REGION Network 4: Block description — Section 3.6 to 4
   // ▂▂▂▂▂▂▂▂▂▂▂▂▂▂▂▂▂▂▂▂▂▂▂▂▂▂▂▂▂▂▂▂▂▂▂▂▂▂▂▂▂▂▂▂
   // 3.6     Operating modes
   // 
   // 
   // This module FC11001_StdDevValveIsol supports various operating modes:
   // 
   //    •   Automatic/manual mode
   // 
   //    •   Interlock bypass mode
   // 
   //    •   Simulation mode
   // 
   //    •   Remote/local mode
   // 
   //    •   Faceplate disabled mode
   // 
   // Examining these in turn:   
   // 
   // 
   // 
   // ▁▁▁▁▁▁▁▁▁▁▁▁▁▁▁▁▁▁▁▁▁▁▁▁▁▁▁▁▁▁▁▁▁▁▁▁▁▁▁▁▁▁▁▁
   // 3.6.1    Automatic and manual modes
   // 
   // 
   // Under normal operation, the valve is in automatic mode and is controlled directly by the 
   // Controller software (usually, sequential or continuous logic); however, it is possible for the 
   // operator to take direct control of the valve by switching it to manual mode.
   // 
   // If manual mode is active, the valve will open and close directly at the command of the operator 
   // and will ignore any automatic mode open and close requests.
   // 
   // If the valve is operating under automatic mode, the manual open/close request follows that of 
   // the automatic mode; this ensures that the valve remains in the same state when initially 
   // switched from automatic mode to manual mode, referred to as bumpless transfer. This approach 
   // minimises any disturbance to the process should the valve be inadvertently switched to manual 
   // mode.
   // 
   // The following data points are associated with automatic/manual mode:
   // 
   //  DATA STRUCTURE    UT11001_St_DevValveIsol
   //  ――――――――――――――――――――――――――――――――――――――――――
   //  SIGNAL         FUNCTION               TYPE     DETAILS
   //  ――――――――――――――――――――――――――――――――――――――――――
   //  CONFIG_MAN_DIS     Prevents manual mode being       Bool  1 = no manual mode
   //            activated under all circumstances            0 = manual permitted
   //  ――――――――――――――――――――――――――――――――――――――――――
   // 
   //  DATA STRUCTURE    UT31001_Dy_DevValveIsol
   //  ――――――――――――――――――――――――――――――――――――――――――
   //  SIGNAL         FUNCTION               TYPE     DETAILS
   //  ――――――――――――――――――――――――――――――――――――――――――
   //  Mode_AutMan     Identifies the operating mode of     Bool  1 = automatic mode
   //            the valve.                   0 = manual mode
   // 
   //  ctrl_Aut_OpenClose Causes the valve to open and close     Bool  1 = open the valve
   //            if automatic mode is active            0 = close the valve
   // 
   //  ctrl_Man_OpenClose  Causes the valve to open and close     Bool  1 = open the valve
   //            if manual mode is active             0 = close the valve
   // 
   //  status_Aut      The valve is in automatic mode      Bool  1 = auto mode
   //                                  0 = no in auto
   // 
   //  status_Man       The valve is in manual mode     Bool  1 = manual mode
   //                                  0 = no in manual
   //  ――――――――――――――――――――――――――――――――――――――――――
   // 
   // Manual mode can only be activated by the operator via a faceplate available at the supervisory 
   // system (SCADA/HMI). 
   // 
   // 
   // 
   // ▁▁▁▁▁▁▁▁▁▁▁▁▁▁▁▁▁▁▁▁▁▁▁▁▁▁▁▁▁▁▁▁▁▁▁▁▁▁▁▁▁▁▁▁
   // 3.6.2    Interlock bypass mode
   // 
   // 
   // All interlock signals (TRIP, INTERLOCK or PERMISSIVE) can be overridden (bypassed). The bypass 
   // signal is a single signal that, if active, overrides and deactivates any TRIP, INTERLOCK or 
   // PERMISSIVE signal that may have been activated.
   // 
   // It is possible to permanently disable the bypass mode for any given valve (preventing the 
   // operator from activating it).
   // 
   // The following data points are associated with the bypass mode:
   // 
   //  DATA STRUCTURE    UT11001_St_DevValveIsol
   //  ――――――――――――――――――――――――――――――――――――――――――
   //  SIGNAL       FUNCTION                TYPE     DETAILS
   //  ――――――――――――――――――――――――――――――――――――――――――
   //  CONFIG_BYPASS_DIS    Prevents bypass mode being      Bool     1 = no bypass mode
   //             activated under all circumstances         0 = bypass permitted
   //  ――――――――――――――――――――――――――――――――――――――――――
   // 
   //  DATA STRUCTURE    UT31001_Dy_DevValveIsol
   //  ――――――――――――――――――――――――――――――――――――――――――
   //  SIGNAL         FUNCTION                TYPE     DETAILS
   //  ――――――――――――――――――――――――――――――――――――――――――
   //  mode_BypassOn   Activates bypass mode, if active, any    Bool     1 = bypass mode on
   //            TRIP, INTERLOCK or PERMISSIVE signal          0 = bypass mode off
   //            will be ignored
   // 
   //  status_BypassOn   Status indication, shows if bypass      Bool     1 = bypass active
   //            mode is active                 0 = bypass inactive
   //  ――――――――――――――――――――――――――――――――――――――――――
   // 
   // Bypass mode can only be activated by the operator usually via a faceplate available at the 
   // supervisory system (SCADA/HMI), alternatively it may be via some form of hardwired signal such 
   // as a key-switch &c. 
   // 
   // If bypass mode is disabled (configuration signal CONFIG_BYPASS_DIS is set to 1), then the bypass 
   // mode cannot be turned on under any circumstances, the option will be greyed out on the 
   // supervisory system faceplate and the module will constantly reset the mode_BypassOn signal.  
   // 
   // 
   // 
   // ▁▁▁▁▁▁▁▁▁▁▁▁▁▁▁▁▁▁▁▁▁▁▁▁▁▁▁▁▁▁▁▁▁▁▁▁▁▁▁▁▁▁▁▁
   // 3.6.3    Simulation mode
   // 
   // 
   // The module can be switched to a simulation mode, in which the position feedback for the valve 
   // is replaced by simulated signals specified by the operator. 
   // 
   // Simulation mode is generally used during testing, but can also be applied in a process 
   // environment if a fault condition is detected; this scenario allows the plant to continue operating 
   // (albeit under some degree of manual control) until the valve is repaired or replaced.
   // 
   // The following data points are associated with the simulation mode:
   // 
   //  DATA STRUCTURE    UT11001_St_DevValveIsol
   //  ――――――――――――――――――――――――――――――――――――――――――
   //  SIGNAL       FUNCTION                TYPE     DETAILS
   //  ――――――――――――――――――――――――――――――――――――――――――
   //  CONFIG_SIM_DIS     Prevents simulation mode being     Bool     1 = no sim mode
   //             activated under all circumstances         0 = sim permitted
   //  ――――――――――――――――――――――――――――――――――――――――――
   // 
   //  DATA STRUCTURE    UT31001_Dy_DevValveIsol
   //  ――――――――――――――――――――――――――――――――――――――――――
   //  SIGNAL         FUNCTION                TYPE     DETAILS
   //  ――――――――――――――――――――――――――――――――――――――――――
   //  mode_SimOn      Activates simulation mode, if active, the   Bool     1 = sim mode on
   //            position feedback will be specified by         0 = sim mode off
   //            mode_SimValue      
   //  mode_SimValue    Specifies the type of simulated position     Int     0 = no feedback
   //            feedback in use                  1 = permanently open
   //                                      2 = permanently closed
   //                                      3 = follow demand
   // 
   //  status_SimOn     Status indication, shows if simulation     Bool     1 = sim active
   //            mode is active                 0 = sim inactive
   //  ――――――――――――――――――――――――――――――――――――――――――
   // 
   // Simulation mode can only be activated by the operator via a faceplate available at the 
   // supervisory system (SCADA/HMI).
   // 
   // If simulation mode is activated, the position feedback for the valve is forced to one of four 
   // states specified by the mode_SimValue variable (this is an enumerated variable):
   // 
   //  ――――――――――――――――――――――――――――――――――――――――――
   //  mode_SimValue  DESCRIPTION               FBK_OPEN FBK_CLOSED
   //  ――――――――――――――――――――――――――――――――――――――――――
   //      0        Permanently disables all position feedback    0     0
   //             (irrespective of any valve position)
   // 
   //      1        Permanently sets valve position to open         1     0
   //             (irrespective of any valve position)
   // 
   //      2        Permanently sets valve position to closed      0     1
   //             (irrespective of any valve position)
   // 
   //      3        Position feedback follows the requested        1/0    0/1
   //             state of the valve              (if valve is open/closed)
   //  ――――――――――――――――――――――――――――――――――――――――――
   // 
   // The mode_SimValue is restricted to the range 0-3.
   // 
   // If simulation mode is disabled (configuration signal CONFIG_SIM_DIS is set to 1), then the 
   // simulation mode cannot be turned on under any circumstances, the option will be greyed out on 
   // the supervisory system faceplate and the module will constantly reset the mode_SimOn signal.
   // 
   // If simulation mode is permitted (CONFIG_SIM_DIS = 0), then setting mode_SimOn to 1 will activate 
   // simulation mode and the any position feedback signals (connected to FBK_OPEN and 
   // FBK_CLOSED) will be overridden according to the value stored in mode_SimValue (see Table above).
   // 
   // The operator can set and adjust the simulation value (mode_SimValue) from the instrument 
   // faceplate on the supervisory system. The simulation value can be adjusted at any time by the 
   // operator (even if simulation mode has not been activated), but will not be applied until 
   // simulation mode is turned on (mode_SimOn = 1). 
   // 
   // If simulation mode is completely disabled (CONFIG_SIM_DIS is set to 1) then the operator will not 
   // be able to adjust the simulated value (mode_SimValue will be greyed out on the faceplate).
   // 
   // 
   // 
   // ▁▁▁▁▁▁▁▁▁▁▁▁▁▁▁▁▁▁▁▁▁▁▁▁▁▁▁▁▁▁▁▁▁▁▁▁▁▁▁▁▁▁▁▁
   // 3.6.4     Remote/local mode
   // 
   // Remote and local operating modes refer to the supervisory system that has control of the 
   // device (i.e. which system can write to the device and change the operating mode of the 
   // device). 
   // 
   // This type of mode is usual present where a plant has a remote central control location (a control 
   // room) that normally controls the device (remote control), but also has a field panel with a local 
   // HMI that an operator in the field can select to take over control of the device (local control) for 
   // maintenance purposes.
   // 
   // The modes are as follows (and are mutually exclusive, only one will be active):
   // 
   //    Remote        Only the remote system in the control room can 
   //                 control the device
   // 
   //    Local            A local system has taken control of the device and the remote 
   //                 system can no longer issue commands to it
   // 
   //    Remote/local disabled   The system does not use remote/local modes and any 
   //      (ALL mode)     supervisory system can issue commands to the device 
   //  
   // Remote/local control is generally handled by the supervisory systems themselves; however, the 
   // supervisory systems need a storage area per device to record which mode that device is in, local 
   // control is often activated by a panel key-switch, that changes the state of several devices from 
   // remote to local (usually all the devices controlled by the local panel).
   // 
   // The module simply identifies the remote/local mode from the mode signals and configuration 
   // signals provided to the module.
   // 
   // For systems that do not use remote/local modes (any supervisory system can control the device, 
   // or control is determined by operator privileges), the remote/local modes can be disabled 
   // (CONFIG_RL_EN is set to zero) and the device is effectively in ALL mode (any system can 
   // control the device).
   // 
   // If remote/local operation is in use, the supervisory system that does not have control will still 
   // display all the information from the device, but will not be able to control the device (it could not 
   // for example, activate simulation mode) and all control function (faceplate functions) will be 
   // greyed out.
   // 
   // The following signals are associated with remote/local/all modes:
   // 
   //  DATA STRUCTURE    UT11001_St_DevValveIsol
   //  ――――――――――――――――――――――――――――――――――――――――――
   //  SIGNAL           FUNCTION            TYPE   DETAILS
   //  ――――――――――――――――――――――――――――――――――――――――――
   //  CONFIG_RL_EN      Allows Remote and Local      Bool    1 = Remote/local selected
   //                 modes to be selected        0 = All mode is active
   // 
   //  DATA STRUCTURE    UT31001_Dy_DevValveIsol
   //  ――――――――――――――――――――――――――――――――――――――――――
   //  SIGNAL           FUNCTION            TYPE   DETAILS
   //  ――――――――――――――――――――――――――――――――――――――――――
   //  mode_RemoteOn       Activates remote mode     Bool    1 = remote mode on, 
   //                 CONFIG_RL_EN must = 1       0 = remote mode off
   // 
   //  mode_LocalOn     Activates local mode          Bool    1 = local mode on, 
   //                 CONFIG_RL_EN must = 1       0 = remote mode off
   // 
   //  status_RemoteOn      Status remote mode on     Bool    1 = remote mode on, 
   //                               0 = remote mode off
   // 
   //  status_LocalOn       Status local mode on      Bool 1 = local mode on, 
   //                               0 = local mode off
   // 
   //  status_RLOff       Status ALL mode is on = 0    Bool 1 = ALL mode on, 
   //                               0 = ALL mode off
   //  ――――――――――――――――――――――――――――――――――――――――――
   //  Block remote/local signals 
   // 
   // By default, remote/local is disabled — ALL mode is selected (CONFIG_RL_EN = 0).
   // 
   // 
   // 
   // 
   // ▁▁▁▁▁▁▁▁▁▁▁▁▁▁▁▁▁▁▁▁▁▁▁▁▁▁▁▁▁▁▁▁▁▁▁▁▁▁▁▁▁▁▁▁
   // 3.6.5     Faceplate disable mode
   // 
   // It is possible to disable the supervisory system faceplate from within the module, the 
   // configuration signal:
   // 
   // 
   //  ――――――――――――――――――――――――――――――――――――――――――
   //  SIGNAL           FUNCTION            TYPE   DETAILS
   //  ――――――――――――――――――――――――――――――――――――――――――
   //  CONFIG_FP_DIS        Disable the supervisory      Bool    1 = Faceplate disabled
   //                 system faceplate           0 = normal
   //  ――――――――――――――――――――――――――――――――――――――――――
   // 
   // If the faceplate is disabled (CONFIG_FP_DIS = 1), the supervisory system must not allow the 
   // device faceplate to be opened (normally achieved by clicking the block icon or device symbol), 
   // this in turn prevents the operator from affecting the device in anyway, it would not, for example, 
   // be possible to put the device into simulation mode.
   // 
   // Similarly, if the faceplate is disabled, the operator will not have access to the mode_Reset signal, 
   // meaning that alternative reset mechanisms must be in place (such as a hardwired pushbutton 
   // for example).
   // 
   //                ━━━   ⬙⬙⬙⬙⬙⬙   ━━━
   // 
   // 
   // 
   // ▄▄▄▄▄▄▄▄▄▄▄▄▄▄▄▄▄▄▄▄▄▄▄▄▄▄▄▄▄▄▄▄▄▄▄▄▄▄▄▄▄▄▄▄
   // 4.     Supervisory system interface
   // 
   // 
   // See the online documentation for this block — select the block in the project tree and press:
   //      SHIFT + F1 or follow the link: https://psop.uk/pal-smds-fc11001-p 
   // 
   // An explanation of the block icons and faceplates available to the supervisory system for this 
   // module is given in section 4 of the SMDS document [Ref. 011].
   // 
   // A downloadable copy of the SMDS (and all other project documentation) is available here:
   // 
   //      https://practicalseries.com/2001-pal/21-project/01-00-docs.html
   // 
   // For this module, the document number is: PS2001-5-2312-fc11001
   // 
   //                ━━━   ⬙⬙⬙⬙⬙⬙   ━━━
END_REGION

REGION Network 5: Block description — Sections 5 to 11
   // ▄▄▄▄▄▄▄▄▄▄▄▄▄▄▄▄▄▄▄▄▄▄▄▄▄▄▄▄▄▄▄▄▄▄▄▄▄▄▄▄▄▄▄▄
   // 5.     PARAMETERS
   // 
   // 
   // The following parameters are associated with the block:
   // 
   //  
   //  ――――――――――――――――――――――――――――――――――――――――――
   //  PARAM         FUNCTION                    TYPE      IN-OUT 
   //  ――――――――――――――――――――――――――――――――――――――――――
   //  SYS_SIGNALS      Common system signals              UT21000    In
   //           logic and timing signals for parametric access
   // 
   //  FBK_OPEN     Optional open state positive feedback        Bool      In
   //           (1 = open, 0 = not open) If not required, set 
   //           permanently to _False
   // 
   //  FBK_CLOSED    Optional closed state positive feedback        Bool      In
   //           (1 = closed 0 = not closed) If not required, set 
   //           permanently to _False
   // 
   //  EXT_FAULT     Optional external fault signal for the device     Bool      In
   //           (1 = fault, 0 = healthy). If not required, set 
   //           permanently to _False
   // 
   //  E_STOP        Optional emergency stop (safety) signal        Bool      In
   //           (1 = emergency stop active, 0 = healthy) If not 
   //           required, set permanently to _False
   // 
   //  TRIP        Optional trip signal                  Bool      In
   //           (1 = trip condition active, 0 = healthy) If not 
   //           required, set permanently to _False
   // 
   //  INTERLOCK     Optional interlock signal               Bool      In
   //           (1 = interlock condition active, 0 = healthy) If 
   //           not required, set permanently to _False
   // 
   //  PERMISSIVE      Optional permissive signal             Bool      In
   //           (1 = permissive condition active, 0 = healthy) 
   //           If not required, set permanently to _False
   // 
   //  STATIC_DATA     Data structure that holds the configuration data     UT11001    In
   //           for the device (normally open/closed, limit switch 
   //           and interlock configuration &c.)
   // 
   //  DYNAMIC_DATA      Data structure that holds the live data for the       UT31001    InOut
   //           device (its mode, status and messages and 
   //           any other dynamic information required by the 
   //           module)
   // 
   //  OPERATE        Output to drive the valve to a particular state    Bool      Out
   //           (1 = energised state, 0 = deenergised state)
   //  ――――――――――――――――――――――――――――――――――――――――――
   // 
   //                ━━━   ⬙⬙⬙⬙⬙⬙   ━━━
   // 
   // 
   // 
   // ▄▄▄▄▄▄▄▄▄▄▄▄▄▄▄▄▄▄▄▄▄▄▄▄▄▄▄▄▄▄▄▄▄▄▄▄▄▄▄▄▄▄▄▄
   // 6.     DATA STRUCTURES AND USAGE
   // 
   // 
   // The block has the following associated data structure:
   // 
   // 
   //  ――――――――――――――――――――――――――――――――――――――――――
   //  DATA STRUCTURE             DESCRIPTION
   //  ――――――――――――――――――――――――――――――――――――――――――
   //  UT01000_St_SysRevision          Revision information for this block    See FC01001
   //  UT01001_St_SysLicence           Licence information for this block  See FC01001
   //  UT21000_Dy_SysSignals           System signals for logic and timing  See FC01001
   // 
   //  UT11001_St_DevValveIsol        Static data that holds the configuration data
   //                     for the device (normally open/closed, limit switch 
   //                     and interlock configuration &c.)
   // 
   //  UT31001_Dy_DevValveIsol          Dynamic data that holds the live data for the
   //                     device (its mode, status and messages and 
   //                     any other dynamic information required by the 
   //                     module)
   // 
   //  ――――――――――――――――――――――――――――――――――――――――――
   // 
   // 
   // 
   // ▂▂▂▂▂▂▂▂▂▂▂▂▂▂▂▂▂▂▂▂▂▂▂▂▂▂▂▂▂▂▂▂▂▂▂▂▂▂▂▂▂▂▂▂
   // 6.1     UT11001_St_DevValveIsol
   // 
   // The static data structure for an isolating valve.
   // 
   // 
   //  UT11001_St_DevValveIsol (full contents)
   //  ――――――――――――――――――――――――――――――――――――――――――
   //  SIGNAL NAME          FUNCTION                     TYPE
   //  ――――――――――――――――――――――――――――――――――――――――――
   //  CONFIG_NO_NC        CONFIG — Normally open or normally closed valve     Bool
   //                      (1 = normally open, 0 = normally closed)
   //  CONFIG_FBK_OPEN_EN    CONFIG — Open feedback is enabled        Bool
   //                      (1 = open feedback, 0 = no feedback)
   //  CONFIG_FBK_CLOSED_EN   CONFIG — Closed feedback is enabled         Bool
   //                      (1 = closed feedback, 0 = no feedback)
   //  CONFIG_ESTOP_DIS     CONFIG — E_STOP signal disabled           Bool
   //                      (1 = E_STOP not used, 0 = in use)
   //  CONFIG_TRIP_DIS      CONFIG — TRIP signal disabled           Bool
   //                      (1 = TRIP not used, 0 = in use)
   //  CONFIG_ILOCK_DIS     CONFIG — INTERLOCK signal disabled        Bool
   //                      (1 = INTERLOCK not used, 0 = in use)
   //  CONFIG_PERM_DIS      CONFIG — PERMISSIVE signal disabled         Bool
   //                      (1 = PERMISSIVE not used, 0 = in use)
   //  CONFIG_TRIP_OP_CL       CONFIG — TRIP state                  Bool
   //                      (1 = open, 0 = close)
   //  CONFIG_ILOCK_OP_CL      CONFIG — INTERLOCK state              Bool
   //                      (1 = open, 0 = close)
   //  CONFIG_PERM_OP_CL       CONFIG — PERMISSIVE permitted state         Bool
   //                      (1 = open, 0 = closed)
   //  CONFIG_FP_DIS               CONFIG — Faceplate is disabled           Bool
   //                      (1 = no Faceplate, 0 = normal)
   //  CONFIG_MAN_DIS              CONFIG — Manual mode is disabled          Bool
   //                      (1 = no manual mode, 0 = normal)
   //  CONFIG_BYPASS_DIS     CONFIG — Bypass mode is disabled           Bool
   //                      (1 = no bypass mode, 0 = normal)
   //  CONFIG_SIM_DIS             CONFIG — Simulation is disabled            Bool
   //                      (1 = no simulation, 0 = normal)
   //  CONFIG_RL_EN       CONFIG — Remote/local mode enabled       Bool
   //                      (1 = enabled, 0 = all mode)
   // 
   //  INFO_TAG          INFORMATION — Instrument ID tag          String[20]
   // 
   //  TIME_OPENING_MAX    TIMER — Initial value of opening operation timer      Real
   //                      (counts down from this value), [seconds]
   //  TIME_CLOSING_MAX       TIMER — Initial value of closing operation timer     Real
   //                      (counts down from this value), [seconds]
   //  TIME_DER_OPEN              TIMER — Percentage of opening timer to expired      Real
   //                      before simulating FBK_OPEN, [percent]
   //  TIME_DER_CLOSED            TIMER — Percentage of closing timer to expired        Real
   //                      before simulating FBK_CLOSED, [percent]
   //  ――――――――――――――――――――――――――――――――――――――――――
   // 
   // 
   // 
   // ▂▂▂▂▂▂▂▂▂▂▂▂▂▂▂▂▂▂▂▂▂▂▂▂▂▂▂▂▂▂▂▂▂▂▂▂▂▂▂▂▂▂▂▂
   // 6.2      UT31001_Dy_DevValveIsol
   // 
   // The static data structure for an isolating valve.
   // 
   // 
   // 
   //  UT31001_Dy_DevValveIsol (full contents)
   //  ――――――――――――――――――――――――――――――――――――――――――
   //  SIGNAL NAME          FUNCTION                     TYPE
   //  ――――――――――――――――――――――――――――――――――――――――――
   //  status_Closed        STATUS — Valve is confirmed closed          Bool
   //                      (1 = closed, 0 = not closed)
   //  status_Open        STATUS — Valve is confirmed open         Bool
   //                      (1 = open, 0 = not open)
   //  status_Closing       STATUS — Valve is closing             Bool
   //                      (1 = closing, 0 = not closing)
   //  status_Opening        STATUS — Valve is opening              Bool
   //                      (1 = opening, 0 = not opening)
   //  status_Operating        STATUS — Valve is changing state           Bool
   //                      (1 = changing state, 0 = fixed state)
   //  status_Fault            STATUS — Valve is in fault              Bool
   //                      (1 = fault present, 0 = healthy)
   //  status_Energised        STATUS — Valve output is on              Bool
   //                      (1 = energised, 0 = deenergised)
   //  status_Aut           STATUS — Automatic mode active           Bool
   //                      (1 = auto mode on, 0 = auto mode off)
   //  status_Man          STATUS — Manual mode active             Bool
   //                      (1 = man mode on, 0 = man mode off)
   //  status_EStop          STATUS — E_STOP safety signal is active         Bool
   //                      (1 = active, 0 = healthy)
   //  status_Trip        STATUS — TRIP signal is active             Bool
   //                      (1 = active, 0 = healthy)
   //  status_Ilock         STATUS — INTERLOCK signal is active            Bool
   //                      (1 = active, 0 = healthy)
   //  status_Perm        STATUS — PERMISSIVE signal is active           Bool
   //                      (1 = active, 0 = healthy)
   //  status_BypassOn        STATUS — Valve is in bypass mode          Bool
   //                      (1 = Simulation mode, 0 = normal)
   //  status_SimOn           STATUS — Valve is in simulation mode               Bool
   //                      (1 = Simulation mode, 0 = normal)
   //  status_RemoteOn       STATUS — Valve is in remote mode                  Bool
   //                      (1 = Remote mode, 0 = normal)
   //  status_LocalOn         STATUS — Valve is in local mode                    Bool
   //                      (1 = Local mode, 0 = normal)
   //  status_RLOff         STATUS — Valve is in ALL mode                   Bool
   //                      (1 = ALL mode, 0 = normal)
   // 
   //  msg_FailToOpen       MESSAGE — Alarm – “Fail to open” is active         Bool
   //  msg_FailToClose       MESSAGE — Alarm – “Fail to close” is active        Bool
   //  msg_FailWhileOpen    MESSAGE — Alarm – “Fail while open” is active      Bool
   //  msg_FailWhileClosed     MESSAGE — Alarm – “Fail while closed” is active   Bool
   //  msg_Flt_External         MESSAGE — Alarm – “external fault" is active      Bool
   // 
   //  mode_AutMan        MODE — Automatic or manual mode selection     Bool
   //                    (1 = auto mode active, 0 = man mode)
   //  mode_BypassOn      MODE — Bypass mode                Bool
   //                    (1 = bypass mode active, 0 = normal)
   //  mode_SimOn         MODE — Simulation mode               Bool
   //                    (1 = sim mode active, 0 = normal)
   //  mode_SimValue       MODE — Simulation value               Int
   //                    (0 = no limits, 1 = always open, 
   //                    2 = always closed, 3 = follow demand)
   //  mode_RemoteOn        MODE — Remote SCADA control enabled       Bool
   //                    (1 = active, 0 = disabled or N/A)
   //  mode_LocalOn         MODE — Local HMI control enabled           Bool
   //                    (1 = active, 0 = disabled or N/A)
   //  mode_Reset        MODE — Fault reset – 1 cycle only           Bool
   //                    (1 = Reset faults, 0 = does nothing)
   //  ctrl_Aut_OpenClose       CONTROL — Auto mode open or close valve     Bool
   //                          (1 = open valve , 0 = close valve)
   //  ctrl_Man_OpenClose      CONTROL — Manual mode open or close valve   Bool
   //                          (1 = open valve , 0 = close valve)
   // 
   //  batch_ID         BATCH — Booking ID (optional for batch operations)   UInt
   // 
   //  actual_Operating_Timer     ACTUAL — Timer value — operating opening/closing  Real
   //                      timer actual value [seconds]
   //  actual_Last_Op_Time       ACTUAL — actual time taken to achieve the last    Real
   //                      good valve position [seconds]
   // 
   //  $derived_fbk_open     INTERNAL — Derived feedback open signal       Bool
   //                          (1 = open , 0 = not open)
   //  $derived_fbk_closed      INTERNAL — Derived feedback closed signal        Bool
   //                          (1 = closed, 0 = not closed)
   //  $sim_fbk_open         INTERNAL — Simulated feedback open signal         Bool
   //                          (1 = open , 0 = not open)
   //  $sim_fbk_closed          INTERNAL — Simulated feedback closed signal      Bool
   //                          (1 = closed, 0 = not closed)
   //  $ctrl_OpenClose       INTERNAL — actual open or close request,         Bool
   //                          incorporates all priorities
   //                         (1 = open valve, 0 = close valve)
   //  $pret_Open             INTERNAL — Edge retention (+ve) rising edge of    Bool
   //                          ctrl_OpenClose (change to opening)
   //  $nret_Close            INTERNAL — Edge retention (-ve) falling edge of        Bool
   //                          ctrl_OpenClose (change to closing)
   //  ――――――――――――――――――――――――――――――――――――――――――
   // 
   // 
   // With the exception of the flowing, all these signals are discussed in the previous sections, the 
   // outstanding items are firstly:
   // 
   //      batch_ID
   // 
   // The batch_ID is not required for normal use; it is only used where a “booking” system is used 
   // (common in batch and routing applications). Such booking applications can acquire the device 
   // if it is free and reserve it for a particular phase of the batch. Batch applications are a topic in 
   // their own right and are discussed separately in the online User Guide.
   // 
   // There are internal working signals (all signals the start with a $ are internal working signals used 
   // by the module). In this instance they are used as follows: 
   //  
   // The $derived_fbk_open and $derived_fbk_closed are the internally derived open and closed 
   // feedback signal used in place of FBK_OPEN and FBK_CLOSED if either CONFIG_FBK_OPEN_EN 
   // or CONFIG_FBK_CLOSED_EN is set to zero.
   // 
   // The $sim_fbk_open and $sim_fbk_closed are the simulated position feedback signal used in 
   // place of FBK_OPEN and FBK_CLOSED if simulation mode is active.
   // 
   // $ctrl_OpenClose is the required state of the valve, it takes into account the auto/manual 
   // requested state and modifies this according to any interlocks, safety signals or faults that 
   // may be present.
   // 
   // The $pret_Open and $nret_Close are edge retention signals used to detect either a rising 
   // (a change to opening) or a falling (a change to closing) edge on the $ctrl_OpenClose signal.
   // 
   // 
   //                ━━━   ⬙⬙⬙⬙⬙⬙   ━━━
   // 
   // 
   // 
   // ▄▄▄▄▄▄▄▄▄▄▄▄▄▄▄▄▄▄▄▄▄▄▄▄▄▄▄▄▄▄▄▄▄▄▄▄▄▄▄▄▄▄▄▄
   // 7.     CONSTANTS AND TEMPORARY (LOCAL) DATA
   // 
   // 
   // 
   // ▂▂▂▂▂▂▂▂▂▂▂▂▂▂▂▂▂▂▂▂▂▂▂▂▂▂▂▂▂▂▂▂▂▂▂▂▂▂▂▂▂▂▂▂
   // 7.1     Constants
   // 
   // 
   // The following constants data is used:
   // 
   //  ――――――――――――――――――――――――――――――――――――――――――
   //  SIGNAL NAME       Value    FUNCTION                  TYPE
   //  ――――――――――――――――――――――――――――――――――――――――――
   //  k_TIME_OP_MIN      0.21      Minimum value for the operation timer     Real
   //  ――――――――――――――――――――――――――――――――――――――――――
   // 
   // 
   // 
   // ▂▂▂▂▂▂▂▂▂▂▂▂▂▂▂▂▂▂▂▂▂▂▂▂▂▂▂▂▂▂▂▂▂▂▂▂▂▂▂▂▂▂▂▂
   // 7.2     Temporary (local) data
   // 
   // 
   // The following temporary data is used:
   // 
   //  ――――――――――――――――――――――――――――――――――――――――――
   //  SIGNAL NAME          FUNCTION                  TYPE
   //  ――――――――――――――――――――――――――――――――――――――――――
   //  revInfo             Revision information for the block         UT01000
   //  licInfo           Licensing information for the block      UT01001
   //  calClosedElapsedTime     Calc - Derived closed signal elapsed time   Real
   //  calOpenElapsedTime       Calc - Derived open signal elapsed time   Real
   //  wrkOpen            Working - open position feedback signal      Bool
   //  wrkClosed         Working - closed position feedback signal   Bool
   //  wrkCtrlPriority40        Working - priority 40 controls the valve      Bool
   //  wrkCtrlPriority30        Working - priority 30 controls the valve      Bool
   //  wrkCtrlPriority20        Working - priority 20 controls the valve      Bool
   //  wrkCtrlPriority10        Working - priority 10 controls the valve      Bool
   //  wrkCtrlPriority00        Working - priority 00 controls the valve      Bool
   //  wrkCtrlAutManOpCl     Working - aut/man open or close request     Bool
   //  wrkTimeFbkOpenSim     Working - Err checked TIME_FBK_OPEN            Real
   //  wrkTimeFbkClosedSim     Working - Err checked TIME_FBK_CLOSED           Real
   //  wrkInt           Working storage area (integer)          Int
   //  wrkReal           Working storage (Real)             Real
   //  wrkDInt           Working storage area (double integer)         DInt
   //  ――――――――――――――――――――――――――――――――――――――――――
   // 
   //                ━━━   ⬙⬙⬙⬙⬙⬙   ━━━
   // 
   // 
   // 
   // ▄▄▄▄▄▄▄▄▄▄▄▄▄▄▄▄▄▄▄▄▄▄▄▄▄▄▄▄▄▄▄▄▄▄▄▄▄▄▄▄▄▄▄▄
   // 8.     BLOCK CALLS AND ASSOCIATIONS
   // 
   // 
   // This section details any blocks which may be called from within this software module (subroutine 
   // functions for example), any partner blocks with which it may be associated (for example a 
   // receive module that is partner with a transmit module &c.). It lists any system functions which 
   // may be called (e.g. reading the real time clock) and any system data types that may be used.
   // 
   // Finally, it lists any special calling requirements for the block (for example, must be called from 
   // within a cyclic interrupt organisation block) and if the block is using “optimised access” (this is 
   // the default arrangement).
   // 
   // 
   // 
   // ▂▂▂▂▂▂▂▂▂▂▂▂▂▂▂▂▂▂▂▂▂▂▂▂▂▂▂▂▂▂▂▂▂▂▂▂▂▂▂▂▂▂▂▂
   // 8.1     Block calls from within this module
   // 
   // 
   // There are no PAL block calls from within this block.
   // 
   // 
   // 
   // ▂▂▂▂▂▂▂▂▂▂▂▂▂▂▂▂▂▂▂▂▂▂▂▂▂▂▂▂▂▂▂▂▂▂▂▂▂▂▂▂▂▂▂▂
   // 8.2     Blocks associated with this module
   // 
   // 
   // This is a stand-alone block and is not associated with any other blocks.
   // 
   // 
   // 
   // ▂▂▂▂▂▂▂▂▂▂▂▂▂▂▂▂▂▂▂▂▂▂▂▂▂▂▂▂▂▂▂▂▂▂▂▂▂▂▂▂▂▂▂▂
   // 8.3     System block calls and system data types
   // 
   // There are no system block calls
   // 
   // 
   // 
   // ▂▂▂▂▂▂▂▂▂▂▂▂▂▂▂▂▂▂▂▂▂▂▂▂▂▂▂▂▂▂▂▂▂▂▂▂▂▂▂▂▂▂▂▂
   // 8.4     Special properties and requirements
   // 
   // 
   // 
   // ▁▁▁▁▁▁▁▁▁▁▁▁▁▁▁▁▁▁▁▁▁▁▁▁▁▁▁▁▁▁▁▁▁▁▁▁▁▁▁▁▁▁▁▁
   // 8.4.1     Block optimisation, IEC compatibility and library conformance
   // 
   // 
   //    •   Block optimisation is ACTIVE for this block.
   // 
   //    •   The block has been checked for IEC compatibility and is compliant.
   // 
   //    •   The block is compatible with all IEC library-conformance module constraints
   // 
   // 
   // 
   // ▁▁▁▁▁▁▁▁▁▁▁▁▁▁▁▁▁▁▁▁▁▁▁▁▁▁▁▁▁▁▁▁▁▁▁▁▁▁▁▁▁▁▁▁
   // 8.4.2     Calling requirements
   // 
   // 
   // There are no special calling requirements for this block.
   // 
   //                ━━━   ⬙⬙⬙⬙⬙⬙   ━━━
   // 
   // 
   // 
   // ▄▄▄▄▄▄▄▄▄▄▄▄▄▄▄▄▄▄▄▄▄▄▄▄▄▄▄▄▄▄▄▄▄▄▄▄▄▄▄▄▄▄▄▄
   // 9.     EXAMPLE USAGE
   // 
   // 
   // The following shows a typical deployment of FC11001:
   // 
   //                         ┌─────────────
   //      ───────────────────┤ FC11001 
   //                         ├───────────────┤
   //    "DB21001_DY_StdGlobalData".SysSignals ─┤ SYS_SIGNALS            %Q1.0
   //                         │             OPERATE ├─  "V001_OPR"
   //                   %I1.2     │               │
   //                 "V001_FBK_OPEN" ─┤ FBK_OPEN             │
   //                         │               │
   //                   %I1.1     │               │
   //               "V001_FBK_CLOSED" ─┤ FBK_CLOSED            │
   //                         │               │
   //            %I1.0            │               │
   //           "V001_FAULT"             │               │
   //        ────┤╱├──────────┤ EXT_FAULT                │
   //                         │               │
   //            %I1.4            │               │
   //          "ZONEA_ESTOP"               │               │
   //        ────┤╱├──────────┤ E_STOP                │
   //                         │               │
   //                    "_False" ─┤ TRIP                    │
   //                         │               │
   //            "DB23002_Dy_ILock.V001"─┤ INTERLOCK             │
   //                         │               │
   //                    "_False" ─┤ PERMISSIVE            │
   //                         │               │
   //                         │               │
   //                         │               │
   //         "DB11001_St_DevValveIsol".V001 ─┤ STATIC_DATA             │
   //                         │
   //         "DB31001_Dy_DevValveIsol".V001 ─┤ DYNAMIC_DATA
   //                         │
   //                         │
   //                                         │
   //                                ─────────┘
   // 
   // 
   //               ━━━   ⬙⬙⬙⬙⬙⬙   ━━━
   // 
   // 
   // 
   // ▄▄▄▄▄▄▄▄▄▄▄▄▄▄▄▄▄▄▄▄▄▄▄▄▄▄▄▄▄▄▄▄▄▄▄▄▄▄▄▄▄▄▄▄
   // 10.     TEST AND VERIFICATION PATH
   // 
   // 
   // The following diagram shows the full test and verification path for the formal release of each 
   // version of the software module. See the Test Plan [Ref. 003] for full details, available here:
   //         https://psop.uk/pal-tp-p
   // 
   // 
   //         FC11001-T001         FC11001-T002
   // 
   //     Test version: 000.801     Test version: 001.801
   //  Released version: 001.000     Released version: 002.000
   // Released commit: D0009    Released commit: D0011
   // 
   //        SCR      SMT              SCV     
   // ＿＿＿＿＿＿┌┐＿＿ ▛▜ ＿＿＿＿＿＿＿＿＿＿＿＿╓╖＿＿
   //       └┘   ▙▟             ╙╜  
   // Initial test           Comments standardised
   // 
   // Initial test to release the      Comments updated & 
   // module following the      minor typographical 
   // development stage.       corrections
   // Full SMT              SCV only
   // 
   // 
   // Where:
   // ――――――――――――――――――――――――――――――――――――――――――――
   //  SCR    Source Code Review      A visual inspection of the software to ensure it has been written  
   // ┌┐             to the correct standards, uses the correct structures within the
   // └┘             software and is generally suitable for deployment.               
   // 
   //  SMT Software Module Test    A full and detailed test of an individual software module in
   //   ▛▜              isolation; such testing requires that all branches of the 
   //   ▙▟              software are tested. 
   // 
   //                It tests all the interfaces to the module, any data recorded or 
   //                stored by the module, all error and exception handling functions 
   //                and tests all timed and interrupt driven operations.
   // 
   //  SCV Software Compatibility     A mechanism for verifying that no executable code software 
   // ╓╖    Verification          changes have been made to a module following changes to
   // ╙╜             comment fields.
   // 
   //                Allows typographical errors &c. to be corrected without forcing 
   //                a full SMT on a module that has not functionally changed.
   // ――――――――――――――――――――――――――――――――――――――――――――
   // 
   // An SCV can only be performed on a module that has at some point previously, successfully 
   // completed both an SCR and SMT. Where an SCV is implemented, it replaces the requirement for 
   // both the SCR and the SMT for the test iteration in question.
   // 
   //                ━━━   ⬙⬙⬙⬙⬙⬙   ━━━
   // 
   // 
   // ██████████████ █ █ █ █  END   █ █ █ █ ██████████████
END_REGION

REGION Network 6: Current revision and modification history
   // ▄▄▄▄▄▄▄▄▄▄▄▄▄▄▄▄▄▄▄▄▄▄▄▄▄▄▄▄▄▄▄▄▄▄▄▄▄▄▄▄▄▄▄▄
   // MODIFICATION HISTORY
   // 
   // 
   // The revision data shown here, in the network comments, contains additional information 
   // reflecting the software development workflow under the version control system (VCS) employed 
   // to track all software changes.
   // 
   // The VCS in use is the Git Source Code Management system in conjunction with the GitHub online 
   // hosting system. The software in its entirety is available in the GitHub remote repository:
   // 
   //      https://github.com/practicalseries/PS2001-pal-software
   // 
   // The repository is public and can be freely copied (forked in GitHub terminology) and used 
   // under the MIT licence. 
   // 
   // The MIT licence is reproduced in full in the last network of this software module.
   // 
   // 
   //  ―――――――――――――――――――――――――――――――――――――――――――
   //  DATE       REVISION             MASTER BRANCH     DEV
   //          (nnn.amm)   COMMIT TAG    (Base ---> Merge)    BRANCH   Author
   //  ———————————————————————————————————————————
   //  2022.04.16    002.000   D0011      D0010 D0011  None    M. Gledhill
   //                        FC11001 — RELEASED FOR USE
   //                          Merge back to master branch
   // 
   //  2022.04.11    001.801   D0010A-000.801   D0010 N/A     D010A   M. Gledhill
   //                        Released for test (SCV)
   // 
   //  2022.04.06    001.101   D0010A-000.104   D0010 N/A     D010A   M. Gledhill
   //                        Comments updated and standardised
   // 
   //  2021.08.23    001.000   D0009      D0008 D0009  None    M. Gledhill
   //                        FC11001 — RELEASED FOR USE
   //                          Merge back to master branch
   // 
   //  2021.08.23    001.000   D0008A-001.000   D0008 N/A     D0008A   M. Gledhill
   //                        FC11001 — Post-test RELEASED FOR USE
   // 
   //  2021.08.17    000.801   D0008A-000.801   D0008 N/A     D0008A   M. Gledhill
   //                        FC11001 Released for SMT
   // 
   //  2021.08.10    000.103   D0008A-000.103   D0008 N/A     D0008A   M. Gledhill
   //                        FC11001 Initial development testing
   // 
   //  2021.07.21    000.102   D0008A-000.102   D0008 N/A     D0008A   M. Gledhill
   //                        FC11001 Incremental build
   // 
   //  2021.07.13    000.101   D0008A-000.101   D0008 N/A     D0008A   M. Gledhill
   //                        FC11001 Block created — Comments added
   //  ———————————————————————————————————————————
   //   Where: nnn  =  Major revision
   //         a  =  Type (1-7 Development, 8 Proving, 9 Qualification, 0 Release)
   //       mm  =  Minor revision (must be 00 if a = 0)
   //         Block properties version number should be set to nn.a (only one decimal place)
   // 
   // ▄▄▄▄▄▄▄▄▄▄▄▄▄▄▄▄▄▄▄▄▄▄▄▄▄▄▄▄▄▄▄▄▄▄▄▄▄▄▄▄▄▄▄▄
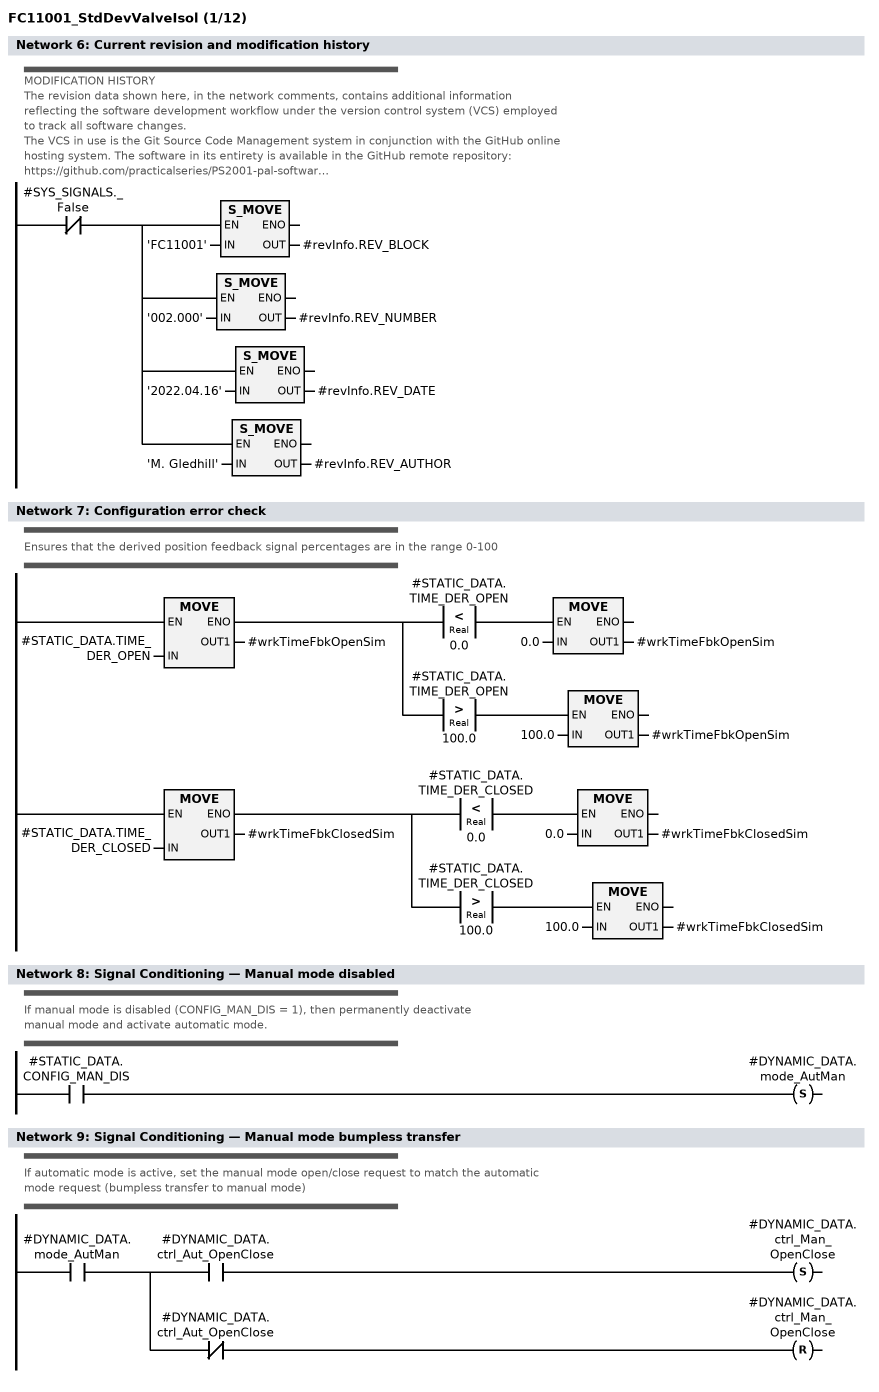
   RUNG wire#powerrail
      I_Contact( #SYS_SIGNALS._False )
      wire#w1
      S_Move(in := 'FC11001', out => #revInfo.REV_BLOCK)
   END_RUNG
   RUNG wire#w1
      S_Move(in := '002.000', out => #revInfo.REV_NUMBER)
   END_RUNG
   RUNG wire#w1
      S_Move(in := '2022.04.16', out => #revInfo.REV_DATE)
   END_RUNG
   RUNG wire#w1
      S_Move(in := 'M. Gledhill', out => #revInfo.REV_AUTHOR)
   END_RUNG
   // the same network as SCL:
   IF NOT #SYS_SIGNALS._False THEN
       #revInfo.REV_BLOCK := 'FC11001';
       #revInfo.REV_NUMBER := '002.000';
       #revInfo.REV_DATE := '2022.04.16';
       #revInfo.REV_AUTHOR := 'M. Gledhill';
   END_IF;
END_REGION

REGION Network 7: Configuration error check
   // ▀▀▀▀▀▀▀▀▀▀▀▀▀▀▀▀▀▀▀▀▀▀▀▀▀▀▀▀▀▀▀▀▀▀▀▀▀▀▀▀▀▀▀▀
   // Ensures that the derived position feedback signal percentages are in the range 0-100
   // ▄▄▄▄▄▄▄▄▄▄▄▄▄▄▄▄▄▄▄▄▄▄▄▄▄▄▄▄▄▄▄▄▄▄▄▄▄▄▄▄▄▄▄▄
   RUNG wire#powerrail
      Move(in := #STATIC_DATA.TIME_DER_OPEN, out1 => #wrkTimeFbkOpenSim)
      wire#w1
      { S7_Templates := "SrcType := Real" } LT_Contact(in1 := #STATIC_DATA.TIME_DER_OPEN, in2 := 0.0)
      Move(in := 0.0, out1 => #wrkTimeFbkOpenSim)
   END_RUNG
   RUNG wire#w1
      { S7_Templates := "SrcType := Real" } GT_Contact(in1 := #STATIC_DATA.TIME_DER_OPEN, in2 := 100.0)
      Move(in := 100.0, out1 => #wrkTimeFbkOpenSim)
   END_RUNG
   RUNG wire#powerrail
      Move(in := #STATIC_DATA.TIME_DER_CLOSED, out1 => #wrkTimeFbkClosedSim)
      wire#w2
      { S7_Templates := "SrcType := Real" } LT_Contact(in1 := #STATIC_DATA.TIME_DER_CLOSED, in2 := 0.0)
      Move(in := 0.0, out1 => #wrkTimeFbkClosedSim)
   END_RUNG
   RUNG wire#w2
      { S7_Templates := "SrcType := Real" } GT_Contact(in1 := #STATIC_DATA.TIME_DER_CLOSED, in2 := 100.0)
      Move(in := 100.0, out1 => #wrkTimeFbkClosedSim)
   END_RUNG
   // the same network as SCL:
   #wrkTimeFbkOpenSim := #STATIC_DATA.TIME_DER_OPEN;
   IF #STATIC_DATA.TIME_DER_OPEN < 0.0 THEN #wrkTimeFbkOpenSim := 0.0; END_IF;
   IF #STATIC_DATA.TIME_DER_OPEN > 100.0 THEN #wrkTimeFbkOpenSim := 100.0; END_IF;
   #wrkTimeFbkClosedSim := #STATIC_DATA.TIME_DER_CLOSED;
   IF #STATIC_DATA.TIME_DER_CLOSED < 0.0 THEN #wrkTimeFbkClosedSim := 0.0; END_IF;
   IF #STATIC_DATA.TIME_DER_CLOSED > 100.0 THEN #wrkTimeFbkClosedSim := 100.0; END_IF;
END_REGION

REGION Network 8: Signal Conditioning — Manual mode disabled
   // ▀▀▀▀▀▀▀▀▀▀▀▀▀▀▀▀▀▀▀▀▀▀▀▀▀▀▀▀▀▀▀▀▀▀▀▀▀▀▀▀▀▀▀▀
   // If manual mode is disabled (CONFIG_MAN_DIS = 1), then permanently deactivate
   // manual mode and activate automatic mode.
   // ▄▄▄▄▄▄▄▄▄▄▄▄▄▄▄▄▄▄▄▄▄▄▄▄▄▄▄▄▄▄▄▄▄▄▄▄▄▄▄▄▄▄▄▄
   RUNG wire#powerrail
      Contact( #STATIC_DATA.CONFIG_MAN_DIS )
      S_Coil( #DYNAMIC_DATA.mode_AutMan )
   END_RUNG
   // the same network as SCL:
   IF #STATIC_DATA.CONFIG_MAN_DIS THEN #DYNAMIC_DATA.mode_AutMan := TRUE; END_IF;
END_REGION

REGION Network 9: Signal Conditioning — Manual mode bumpless transfer
   // ▀▀▀▀▀▀▀▀▀▀▀▀▀▀▀▀▀▀▀▀▀▀▀▀▀▀▀▀▀▀▀▀▀▀▀▀▀▀▀▀▀▀▀▀
   // If automatic mode is active, set the manual mode open/close request to match the automatic
   // mode request (bumpless transfer to manual mode)
   // ▄▄▄▄▄▄▄▄▄▄▄▄▄▄▄▄▄▄▄▄▄▄▄▄▄▄▄▄▄▄▄▄▄▄▄▄▄▄▄▄▄▄▄▄
   RUNG wire#powerrail
      Contact( #DYNAMIC_DATA.mode_AutMan )
      wire#w1
      Contact( #DYNAMIC_DATA.ctrl_Aut_OpenClose )
      S_Coil( #DYNAMIC_DATA.ctrl_Man_OpenClose )
   END_RUNG
   RUNG wire#w1
      I_Contact( #DYNAMIC_DATA.ctrl_Aut_OpenClose )
      R_Coil( #DYNAMIC_DATA.ctrl_Man_OpenClose )
   END_RUNG
   // the same network as SCL:
   IF #DYNAMIC_DATA.mode_AutMan AND #DYNAMIC_DATA.ctrl_Aut_OpenClose THEN
       #DYNAMIC_DATA.ctrl_Man_OpenClose := TRUE;
   END_IF;
   IF #DYNAMIC_DATA.mode_AutMan AND NOT #DYNAMIC_DATA.ctrl_Aut_OpenClose THEN
       #DYNAMIC_DATA.ctrl_Man_OpenClose := FALSE;
   END_IF;
END_REGION

REGION Network 10: Signal Conditioning — Bypass mode disabled
   // ▀▀▀▀▀▀▀▀▀▀▀▀▀▀▀▀▀▀▀▀▀▀▀▀▀▀▀▀▀▀▀▀▀▀▀▀▀▀▀▀▀▀▀▀
   // If bypass mode is disabled (CONFIG_BYPASS_DIS = 1), then permanently deactivate
   // bypass mode.
   // ▄▄▄▄▄▄▄▄▄▄▄▄▄▄▄▄▄▄▄▄▄▄▄▄▄▄▄▄▄▄▄▄▄▄▄▄▄▄▄▄▄▄▄▄
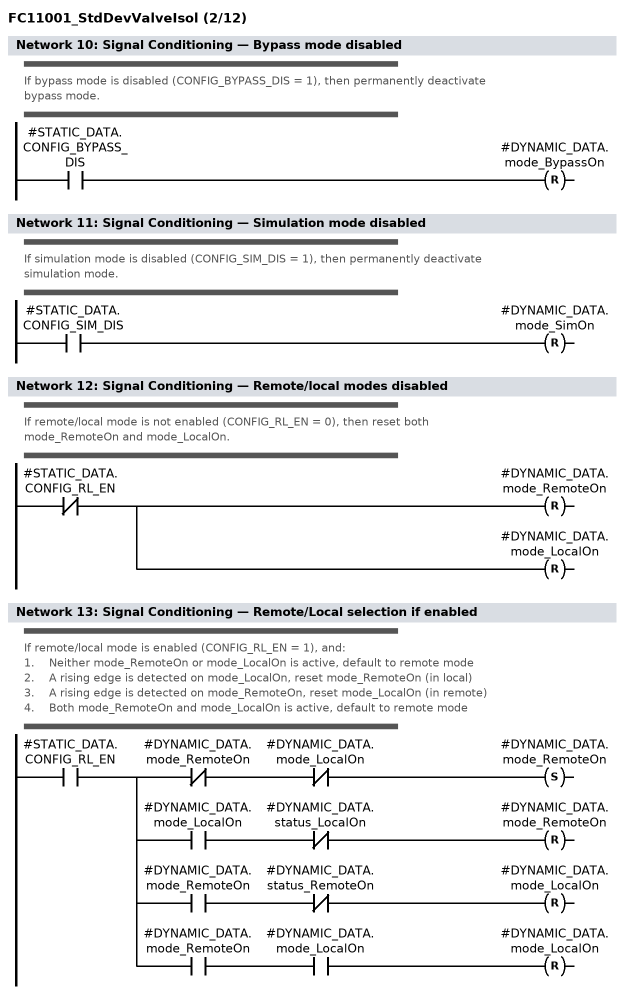
   RUNG wire#powerrail
      Contact( #STATIC_DATA.CONFIG_BYPASS_DIS )
      R_Coil( #DYNAMIC_DATA.mode_BypassOn )
   END_RUNG
   // the same network as SCL:
   IF #STATIC_DATA.CONFIG_BYPASS_DIS THEN #DYNAMIC_DATA.mode_BypassOn := FALSE; END_IF;
END_REGION

REGION Network 11: Signal Conditioning — Simulation mode disabled
   // ▀▀▀▀▀▀▀▀▀▀▀▀▀▀▀▀▀▀▀▀▀▀▀▀▀▀▀▀▀▀▀▀▀▀▀▀▀▀▀▀▀▀▀▀
   // If simulation mode is disabled (CONFIG_SIM_DIS = 1), then permanently deactivate
   // simulation mode.
   // ▄▄▄▄▄▄▄▄▄▄▄▄▄▄▄▄▄▄▄▄▄▄▄▄▄▄▄▄▄▄▄▄▄▄▄▄▄▄▄▄▄▄▄▄
   RUNG wire#powerrail
      Contact( #STATIC_DATA.CONFIG_SIM_DIS )
      R_Coil( #DYNAMIC_DATA.mode_SimOn )
   END_RUNG
   // the same network as SCL:
   IF #STATIC_DATA.CONFIG_SIM_DIS THEN #DYNAMIC_DATA.mode_SimOn := FALSE; END_IF;
END_REGION

REGION Network 12: Signal Conditioning — Remote/local modes disabled
   // ▀▀▀▀▀▀▀▀▀▀▀▀▀▀▀▀▀▀▀▀▀▀▀▀▀▀▀▀▀▀▀▀▀▀▀▀▀▀▀▀▀▀▀▀
   // If remote/local mode is not enabled (CONFIG_RL_EN = 0), then reset both 
   // mode_RemoteOn and mode_LocalOn.
   // ▄▄▄▄▄▄▄▄▄▄▄▄▄▄▄▄▄▄▄▄▄▄▄▄▄▄▄▄▄▄▄▄▄▄▄▄▄▄▄▄▄▄▄▄
   RUNG wire#powerrail
      I_Contact( #STATIC_DATA.CONFIG_RL_EN )
      wire#w1
      R_Coil( #DYNAMIC_DATA.mode_RemoteOn )
   END_RUNG
   RUNG wire#w1
      R_Coil( #DYNAMIC_DATA.mode_LocalOn )
   END_RUNG
   // the same network as SCL:
   IF NOT #STATIC_DATA.CONFIG_RL_EN THEN
       #DYNAMIC_DATA.mode_RemoteOn := FALSE;
       #DYNAMIC_DATA.mode_LocalOn := FALSE;
   END_IF;
END_REGION

REGION Network 13: Signal Conditioning — Remote/Local selection if enabled
   // ▀▀▀▀▀▀▀▀▀▀▀▀▀▀▀▀▀▀▀▀▀▀▀▀▀▀▀▀▀▀▀▀▀▀▀▀▀▀▀▀▀▀▀▀
   // If remote/local mode is enabled (CONFIG_RL_EN = 1), and:
   // 
   //    1.  Neither mode_RemoteOn or mode_LocalOn is active, default to remote mode
   //    2.  A rising edge is detected on mode_LocalOn, reset mode_RemoteOn (in local)
   //    3.  A rising edge is detected on mode_RemoteOn, reset mode_LocalOn (in remote)
   //    4.  Both mode_RemoteOn and mode_LocalOn is active, default to remote mode
   // ▄▄▄▄▄▄▄▄▄▄▄▄▄▄▄▄▄▄▄▄▄▄▄▄▄▄▄▄▄▄▄▄▄▄▄▄▄▄▄▄▄▄▄▄
   RUNG wire#powerrail
      Contact( #STATIC_DATA.CONFIG_RL_EN )
      wire#w1
      I_Contact( #DYNAMIC_DATA.mode_RemoteOn )
      I_Contact( #DYNAMIC_DATA.mode_LocalOn )
      S_Coil( #DYNAMIC_DATA.mode_RemoteOn )
   END_RUNG
   RUNG wire#w1
      Contact( #DYNAMIC_DATA.mode_LocalOn )
      I_Contact( #DYNAMIC_DATA.status_LocalOn )
      R_Coil( #DYNAMIC_DATA.mode_RemoteOn )
   END_RUNG
   RUNG wire#w1
      Contact( #DYNAMIC_DATA.mode_RemoteOn )
      I_Contact( #DYNAMIC_DATA.status_RemoteOn )
      R_Coil( #DYNAMIC_DATA.mode_LocalOn )
   END_RUNG
   RUNG wire#w1
      Contact( #DYNAMIC_DATA.mode_RemoteOn )
      Contact( #DYNAMIC_DATA.mode_LocalOn )
      R_Coil( #DYNAMIC_DATA.mode_LocalOn )
   END_RUNG
   // the same network as SCL:
   IF #STATIC_DATA.CONFIG_RL_EN AND NOT #DYNAMIC_DATA.mode_RemoteOn AND NOT #DYNAMIC_DATA.mode_LocalOn THEN
       #DYNAMIC_DATA.mode_RemoteOn := TRUE;
   END_IF;
   IF #STATIC_DATA.CONFIG_RL_EN AND #DYNAMIC_DATA.mode_LocalOn AND NOT #DYNAMIC_DATA.status_LocalOn THEN
       #DYNAMIC_DATA.mode_RemoteOn := FALSE;
   END_IF;
   IF #STATIC_DATA.CONFIG_RL_EN AND #DYNAMIC_DATA.mode_RemoteOn AND NOT #DYNAMIC_DATA.status_RemoteOn THEN
       #DYNAMIC_DATA.mode_LocalOn := FALSE;
   END_IF;
   IF #STATIC_DATA.CONFIG_RL_EN AND #DYNAMIC_DATA.mode_RemoteOn AND #DYNAMIC_DATA.mode_LocalOn THEN
       #DYNAMIC_DATA.mode_LocalOn := FALSE;
   END_IF;
END_REGION

REGION Network 14: Signal Conditioning — Derived open position
   // ▀▀▀▀▀▀▀▀▀▀▀▀▀▀▀▀▀▀▀▀▀▀▀▀▀▀▀▀▀▀▀▀▀▀▀▀▀▀▀▀▀▀▀▀
   // If there is no open position feedback (CONFIG_FBK_OPEN_EN = 0), then the open state of the 
   // valve is derived from the elapsed time of the operation timer using the following formulae:
   // 
   // ┌───────────────────────────────────────────┐
   // │$derived_fbk_open =1 when:                                │
   // │                                 wrkTimeFbkOpenSim  │
   // │actual_Operating_Timer ≤ TIME_OPENING_MAX ─ TIME_OPENING_MAX ╳ ----------------------------------------│
   // │                                     100     │
   // └───────────────────────────────────────────┘
   // Note:    wrkTimeFbkOpenSim is the error checked equivalent of TIME_FBK_OPEN
   // 
   // If the calculated elapsed time is close to or less than k_TIME_OP_MIN (210ms),
   // the calculated elapsed time (calOpenElapsedTime) is set to k_TIME_OP_MIN. This ensures at
   // least one timing pulse is required before the timer reaches zero.
   // 
   // The derived open signal ($derived_fbk_open) is reset if the valve is requested to be closed
   // ($ctrl_OpenClose = 0).
   // ▄▄▄▄▄▄▄▄▄▄▄▄▄▄▄▄▄▄▄▄▄▄▄▄▄▄▄▄▄▄▄▄▄▄▄▄▄▄▄▄▄▄▄▄
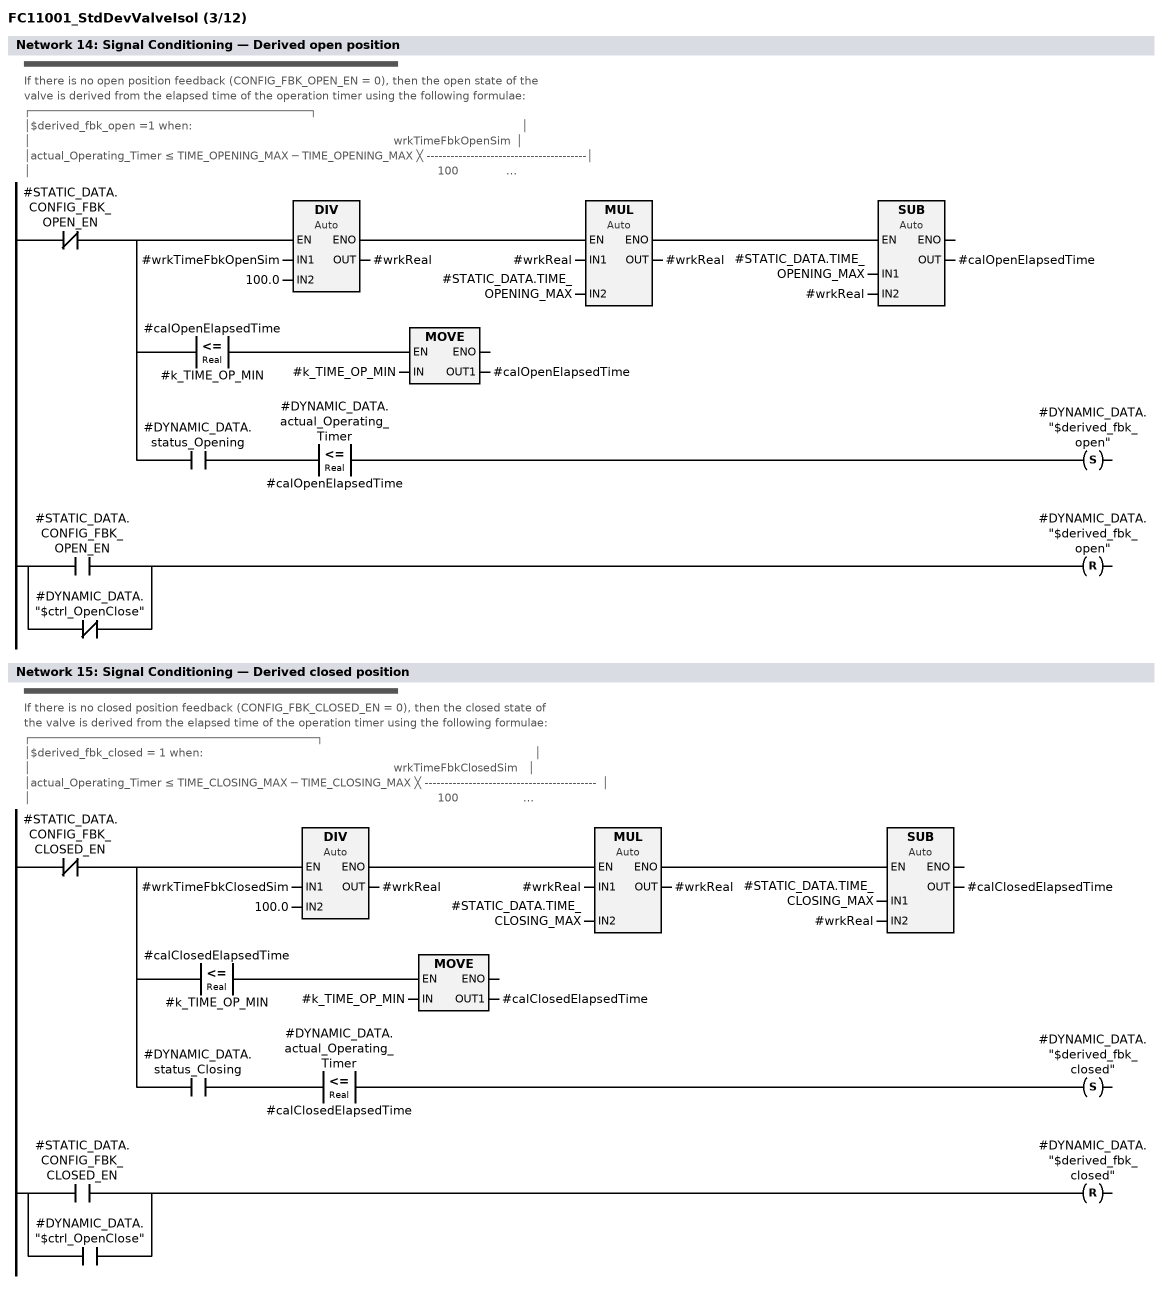
   RUNG wire#powerrail
      I_Contact( #STATIC_DATA.CONFIG_FBK_OPEN_EN )
      wire#w1
      Div(in1 := #wrkTimeFbkOpenSim, in2 := 100.0, out => #wrkReal)
      Mul(in1 := #wrkReal, in2 := #STATIC_DATA.TIME_OPENING_MAX, out => #wrkReal)
      Sub(in1 := #STATIC_DATA.TIME_OPENING_MAX, in2 := #wrkReal, out => #calOpenElapsedTime)
   END_RUNG
   RUNG wire#w1
      { S7_Templates := "SrcType := Real" } LE_Contact(in1 := #calOpenElapsedTime, in2 := #k_TIME_OP_MIN)
      Move(in := #k_TIME_OP_MIN, out1 => #calOpenElapsedTime)
   END_RUNG
   RUNG wire#w1
      Contact( #DYNAMIC_DATA.status_Opening )
      { S7_Templates := "SrcType := Real" } LE_Contact(in1 := #DYNAMIC_DATA.actual_Operating_Timer, in2 := #calOpenElapsedTime)
      S_Coil( #DYNAMIC_DATA."$derived_fbk_open" )
   END_RUNG
   RUNG wire#powerrail
      Contact( #STATIC_DATA.CONFIG_FBK_OPEN_EN )
      wire#w2
      R_Coil( #DYNAMIC_DATA."$derived_fbk_open" )
   END_RUNG
   RUNG wire#powerrail
      I_Contact( #DYNAMIC_DATA."$ctrl_OpenClose" )
   END_RUNG wire#w2
   // the same network as SCL:
   #_w1 := NOT #STATIC_DATA.CONFIG_FBK_OPEN_EN;
   IF #_w1 THEN
       #wrkReal := #wrkTimeFbkOpenSim / 100.0;
       #wrkReal := #wrkReal * #STATIC_DATA.TIME_OPENING_MAX;
       #calOpenElapsedTime := #STATIC_DATA.TIME_OPENING_MAX - #wrkReal;
   END_IF;
   IF #_w1 AND (#calOpenElapsedTime <= #k_TIME_OP_MIN) THEN #calOpenElapsedTime := #k_TIME_OP_MIN; END_IF;
   IF #_w1 AND #DYNAMIC_DATA.status_Opening AND (#DYNAMIC_DATA.actual_Operating_Timer <= #calOpenElapsedTime) THEN
       #DYNAMIC_DATA."$derived_fbk_open" := TRUE;
   END_IF;
   IF #STATIC_DATA.CONFIG_FBK_OPEN_EN OR NOT #DYNAMIC_DATA."$ctrl_OpenClose" THEN
       #DYNAMIC_DATA."$derived_fbk_open" := FALSE;
   END_IF;
END_REGION

REGION Network 15: Signal Conditioning — Derived closed position
   // ▀▀▀▀▀▀▀▀▀▀▀▀▀▀▀▀▀▀▀▀▀▀▀▀▀▀▀▀▀▀▀▀▀▀▀▀▀▀▀▀▀▀▀▀
   // If there is no closed position feedback (CONFIG_FBK_CLOSED_EN = 0), then the closed state of 
   // the valve is derived from the elapsed time of the operation timer using the following formulae:
   // 
   // ┌────────────────────────────────────────────┐
   // │$derived_fbk_closed = 1 when:                                 │
   // │                                 wrkTimeFbkClosedSim   │
   // │actual_Operating_Timer ≤ TIME_CLOSING_MAX ─ TIME_CLOSING_MAX ╳ -------------------------------------------  │
   // │                                     100            │
   // └────────────────────────────────────────────┘
   // Note:    wrkTimeFbkClosedSim is the error checked equivalent of TIME_FBK_CLOSED
   // 
   // If the calculated elapsed time is close to or less than k_TIME_OP_MIN (210ms),
   // the calculated elapsed time (calClosedElapsedTime) is set to k_TIME_OP_MIN. This ensures at
   // least one timing pulse is required before the timer reaches zero.
   // 
   // The derived closed signal ($derived_fbk_closed) is reset if the valve is requested to be open
   // ($ctrl_OpenClose = 1).
   // ▄▄▄▄▄▄▄▄▄▄▄▄▄▄▄▄▄▄▄▄▄▄▄▄▄▄▄▄▄▄▄▄▄▄▄▄▄▄▄▄▄▄▄▄
   RUNG wire#powerrail
      I_Contact( #STATIC_DATA.CONFIG_FBK_CLOSED_EN )
      wire#w1
      Div(in1 := #wrkTimeFbkClosedSim, in2 := 100.0, out => #wrkReal)
      Mul(in1 := #wrkReal, in2 := #STATIC_DATA.TIME_CLOSING_MAX, out => #wrkReal)
      Sub(in1 := #STATIC_DATA.TIME_CLOSING_MAX, in2 := #wrkReal, out => #calClosedElapsedTime)
   END_RUNG
   RUNG wire#w1
      { S7_Templates := "SrcType := Real" } LE_Contact(in1 := #calClosedElapsedTime, in2 := #k_TIME_OP_MIN)
      Move(in := #k_TIME_OP_MIN, out1 => #calClosedElapsedTime)
   END_RUNG
   RUNG wire#w1
      Contact( #DYNAMIC_DATA.status_Closing )
      { S7_Templates := "SrcType := Real" } LE_Contact(in1 := #DYNAMIC_DATA.actual_Operating_Timer, in2 := #calClosedElapsedTime)
      S_Coil( #DYNAMIC_DATA."$derived_fbk_closed" )
   END_RUNG
   RUNG wire#powerrail
      Contact( #STATIC_DATA.CONFIG_FBK_CLOSED_EN )
      wire#w2
      R_Coil( #DYNAMIC_DATA."$derived_fbk_closed" )
   END_RUNG
   RUNG wire#powerrail
      Contact( #DYNAMIC_DATA."$ctrl_OpenClose" )
   END_RUNG wire#w2
   // the same network as SCL:
   #_w1 := NOT #STATIC_DATA.CONFIG_FBK_CLOSED_EN;
   IF #_w1 THEN
       #wrkReal := #wrkTimeFbkClosedSim / 100.0;
       #wrkReal := #wrkReal * #STATIC_DATA.TIME_CLOSING_MAX;
       #calClosedElapsedTime := #STATIC_DATA.TIME_CLOSING_MAX - #wrkReal;
   END_IF;
   IF #_w1 AND (#calClosedElapsedTime <= #k_TIME_OP_MIN) THEN
       #calClosedElapsedTime := #k_TIME_OP_MIN;
   END_IF;
   IF #_w1 AND #DYNAMIC_DATA.status_Closing AND (#DYNAMIC_DATA.actual_Operating_Timer <= #calClosedElapsedTime) THEN
       #DYNAMIC_DATA."$derived_fbk_closed" := TRUE;
   END_IF;
   IF #STATIC_DATA.CONFIG_FBK_CLOSED_EN OR #DYNAMIC_DATA."$ctrl_OpenClose" THEN
       #DYNAMIC_DATA."$derived_fbk_closed" := FALSE;
   END_IF;
END_REGION

REGION Network 16: Signal Conditioning — Simulation mode — Open signal
   // ▀▀▀▀▀▀▀▀▀▀▀▀▀▀▀▀▀▀▀▀▀▀▀▀▀▀▀▀▀▀▀▀▀▀▀▀▀▀▀▀▀▀▀▀
   // If simulation mode is active, the simulated open position signal is set as follows:
   // 
   //    •   mode_SimValue = 0 (no feedback), $sim_fbk_open = 0
   // 
   //    •   mode_SimValue = 1 (permanently open), $sim_fbk_open = 1
   // 
   //    •   mode_SimValue = 2 (permanently closed), $sim_fbk_open = 0
   // 
   //    •   mode_SimValue = 3 (follow demand), $sim_fbk_open = $ctrl_OpenClose
   // 
   // If simulation mode is not active,  $sim_fbk_open = 0
   // ▄▄▄▄▄▄▄▄▄▄▄▄▄▄▄▄▄▄▄▄▄▄▄▄▄▄▄▄▄▄▄▄▄▄▄▄▄▄▄▄▄▄▄▄
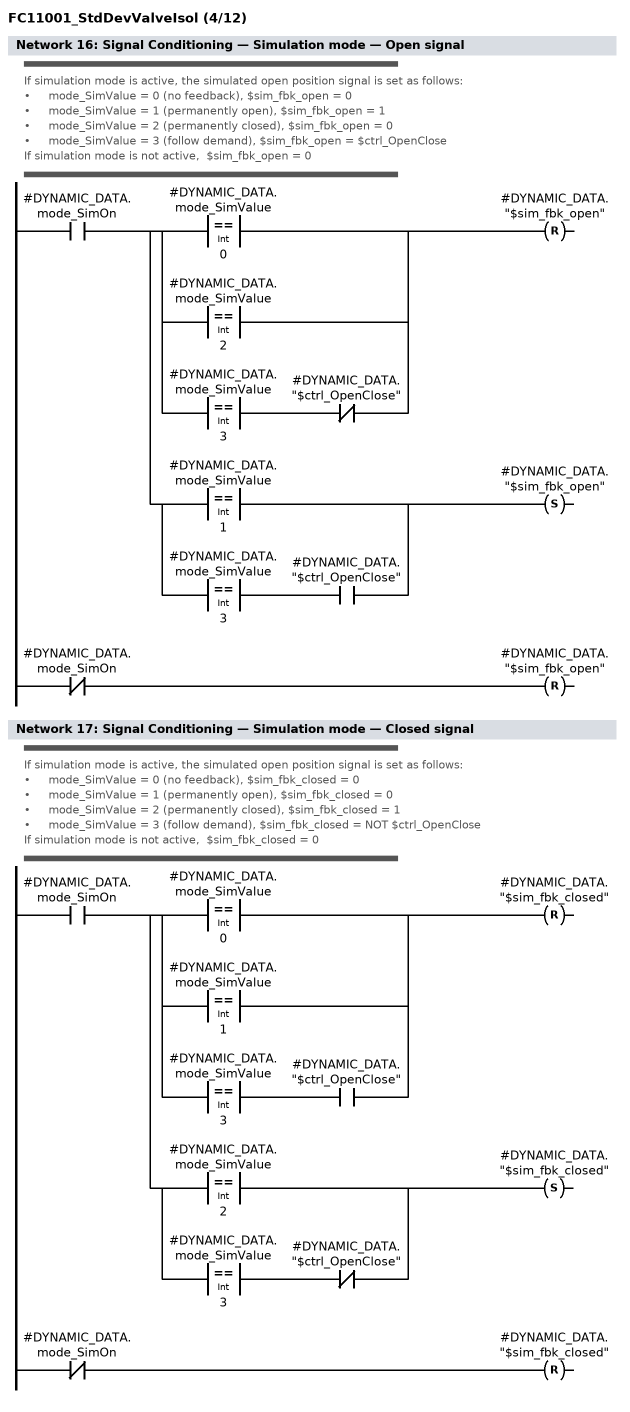
   RUNG wire#powerrail
      Contact( #DYNAMIC_DATA.mode_SimOn )
      wire#w1
      { S7_Templates := "SrcType := Int" } EQ_Contact(in1 := #DYNAMIC_DATA.mode_SimValue, in2 := 0)
      wire#w2
      R_Coil( #DYNAMIC_DATA."$sim_fbk_open" )
   END_RUNG
   RUNG wire#w1
      { S7_Templates := "SrcType := Int" } EQ_Contact(in1 := #DYNAMIC_DATA.mode_SimValue, in2 := 2)
   END_RUNG wire#w2
   RUNG wire#w1
      { S7_Templates := "SrcType := Int" } EQ_Contact(in1 := #DYNAMIC_DATA.mode_SimValue, in2 := 3)
      I_Contact( #DYNAMIC_DATA."$ctrl_OpenClose" )
   END_RUNG wire#w2
   RUNG wire#w1
      { S7_Templates := "SrcType := Int" } EQ_Contact(in1 := #DYNAMIC_DATA.mode_SimValue, in2 := 1)
      wire#w3
      S_Coil( #DYNAMIC_DATA."$sim_fbk_open" )
   END_RUNG
   RUNG wire#w1
      { S7_Templates := "SrcType := Int" } EQ_Contact(in1 := #DYNAMIC_DATA.mode_SimValue, in2 := 3)
      Contact( #DYNAMIC_DATA."$ctrl_OpenClose" )
   END_RUNG wire#w3
   RUNG wire#powerrail
      I_Contact( #DYNAMIC_DATA.mode_SimOn )
      R_Coil( #DYNAMIC_DATA."$sim_fbk_open" )
   END_RUNG
   // the same network as SCL:
   IF #DYNAMIC_DATA.mode_SimOn AND ((#DYNAMIC_DATA.mode_SimValue = 0) OR (#DYNAMIC_DATA.mode_SimValue = 2) OR ((#DYNAMIC_DATA.mode_SimValue = 3) AND NOT #DYNAMIC_DATA."$ctrl_OpenClose")) THEN
       #DYNAMIC_DATA."$sim_fbk_open" := FALSE;
   END_IF;
   IF #DYNAMIC_DATA.mode_SimOn AND ((#DYNAMIC_DATA.mode_SimValue = 1) OR ((#DYNAMIC_DATA.mode_SimValue = 3) AND #DYNAMIC_DATA."$ctrl_OpenClose")) THEN
       #DYNAMIC_DATA."$sim_fbk_open" := TRUE;
   END_IF;
   IF NOT #DYNAMIC_DATA.mode_SimOn THEN #DYNAMIC_DATA."$sim_fbk_open" := FALSE; END_IF;
END_REGION

REGION Network 17: Signal Conditioning — Simulation mode — Closed signal
   // ▀▀▀▀▀▀▀▀▀▀▀▀▀▀▀▀▀▀▀▀▀▀▀▀▀▀▀▀▀▀▀▀▀▀▀▀▀▀▀▀▀▀▀▀
   // If simulation mode is active, the simulated open position signal is set as follows:
   // 
   //    •   mode_SimValue = 0 (no feedback), $sim_fbk_closed = 0
   // 
   //    •   mode_SimValue = 1 (permanently open), $sim_fbk_closed = 0
   // 
   //    •   mode_SimValue = 2 (permanently closed), $sim_fbk_closed = 1
   // 
   //    •   mode_SimValue = 3 (follow demand), $sim_fbk_closed = NOT $ctrl_OpenClose
   // 
   // If simulation mode is not active,  $sim_fbk_closed = 0
   // ▄▄▄▄▄▄▄▄▄▄▄▄▄▄▄▄▄▄▄▄▄▄▄▄▄▄▄▄▄▄▄▄▄▄▄▄▄▄▄▄▄▄▄▄
   RUNG wire#powerrail
      Contact( #DYNAMIC_DATA.mode_SimOn )
      wire#w1
      { S7_Templates := "SrcType := Int" } EQ_Contact(in1 := #DYNAMIC_DATA.mode_SimValue, in2 := 0)
      wire#w2
      R_Coil( #DYNAMIC_DATA."$sim_fbk_closed" )
   END_RUNG
   RUNG wire#w1
      { S7_Templates := "SrcType := Int" } EQ_Contact(in1 := #DYNAMIC_DATA.mode_SimValue, in2 := 1)
   END_RUNG wire#w2
   RUNG wire#w1
      { S7_Templates := "SrcType := Int" } EQ_Contact(in1 := #DYNAMIC_DATA.mode_SimValue, in2 := 3)
      Contact( #DYNAMIC_DATA."$ctrl_OpenClose" )
   END_RUNG wire#w2
   RUNG wire#w1
      { S7_Templates := "SrcType := Int" } EQ_Contact(in1 := #DYNAMIC_DATA.mode_SimValue, in2 := 2)
      wire#w3
      S_Coil( #DYNAMIC_DATA."$sim_fbk_closed" )
   END_RUNG
   RUNG wire#w1
      { S7_Templates := "SrcType := Int" } EQ_Contact(in1 := #DYNAMIC_DATA.mode_SimValue, in2 := 3)
      I_Contact( #DYNAMIC_DATA."$ctrl_OpenClose" )
   END_RUNG wire#w3
   RUNG wire#powerrail
      I_Contact( #DYNAMIC_DATA.mode_SimOn )
      R_Coil( #DYNAMIC_DATA."$sim_fbk_closed" )
   END_RUNG
   // the same network as SCL:
   IF #DYNAMIC_DATA.mode_SimOn AND ((#DYNAMIC_DATA.mode_SimValue = 0) OR (#DYNAMIC_DATA.mode_SimValue = 1) OR ((#DYNAMIC_DATA.mode_SimValue = 3) AND #DYNAMIC_DATA."$ctrl_OpenClose")) THEN
       #DYNAMIC_DATA."$sim_fbk_closed" := FALSE;
   END_IF;
   IF #DYNAMIC_DATA.mode_SimOn AND ((#DYNAMIC_DATA.mode_SimValue = 2) OR ((#DYNAMIC_DATA.mode_SimValue = 3) AND NOT #DYNAMIC_DATA."$ctrl_OpenClose")) THEN
       #DYNAMIC_DATA."$sim_fbk_closed" := TRUE;
   END_IF;
   IF NOT #DYNAMIC_DATA.mode_SimOn THEN #DYNAMIC_DATA."$sim_fbk_closed" := FALSE; END_IF;
END_REGION

REGION Network 18: Signal conditioning — Determine valve OPEN position status
   // ▀▀▀▀▀▀▀▀▀▀▀▀▀▀▀▀▀▀▀▀▀▀▀▀▀▀▀▀▀▀▀▀▀▀▀▀▀▀▀▀▀▀▀▀
   // Generates a working open signal (wrkOpen), that is then used throughout the module as the 
   // definitive open position feedback signal.
   // 
   // The open signal will be either :
   // 
   //    1.  The same as the FBK_OPEN parameter if this is in use 
   //      (CONFIG_FBK_OPEN_EN = 1)
   // 
   //    2.  The internally derived open state (based on the requested state of the valve) if the 
   //      FBK_OPEN signal is NOT in use (CONFIG_FBK_OPEN_EN = 0)
   // 
   //    3.  The simulated state of the valve if simulation mode is active (mode_SimOn = 1)
   // 
   // If an actual open position signal is provided to the module via the FBK_OPEN parameter 
   // (i.e. if CONFIG_FBK_OPEN_EN = 1) then wrkOpen is set to match the FBK_OPEN signal 
   // (wrkOpen = FBK_OPEN).
   // 
   // If a derived open signal is to be used (i.e. if CONFIG_FBK_OPEN_EN = 0), then wrkOpen is set to 
   // match the internally derived $derived_fbk_open signal (wrkOpen = $derived_fbk_open). 
   // $derived_fbk_open is based on the requested state of the valve. 
   // 
   // Finally, if simulation mode is active (mode_SimOn = 1), then wrkOpen is set to match the internal 
   // simulation signal $sim_fbk_open signal (wrkOpen = $sim_fbk_open).. 
   // ▄▄▄▄▄▄▄▄▄▄▄▄▄▄▄▄▄▄▄▄▄▄▄▄▄▄▄▄▄▄▄▄▄▄▄▄▄▄▄▄▄▄▄▄
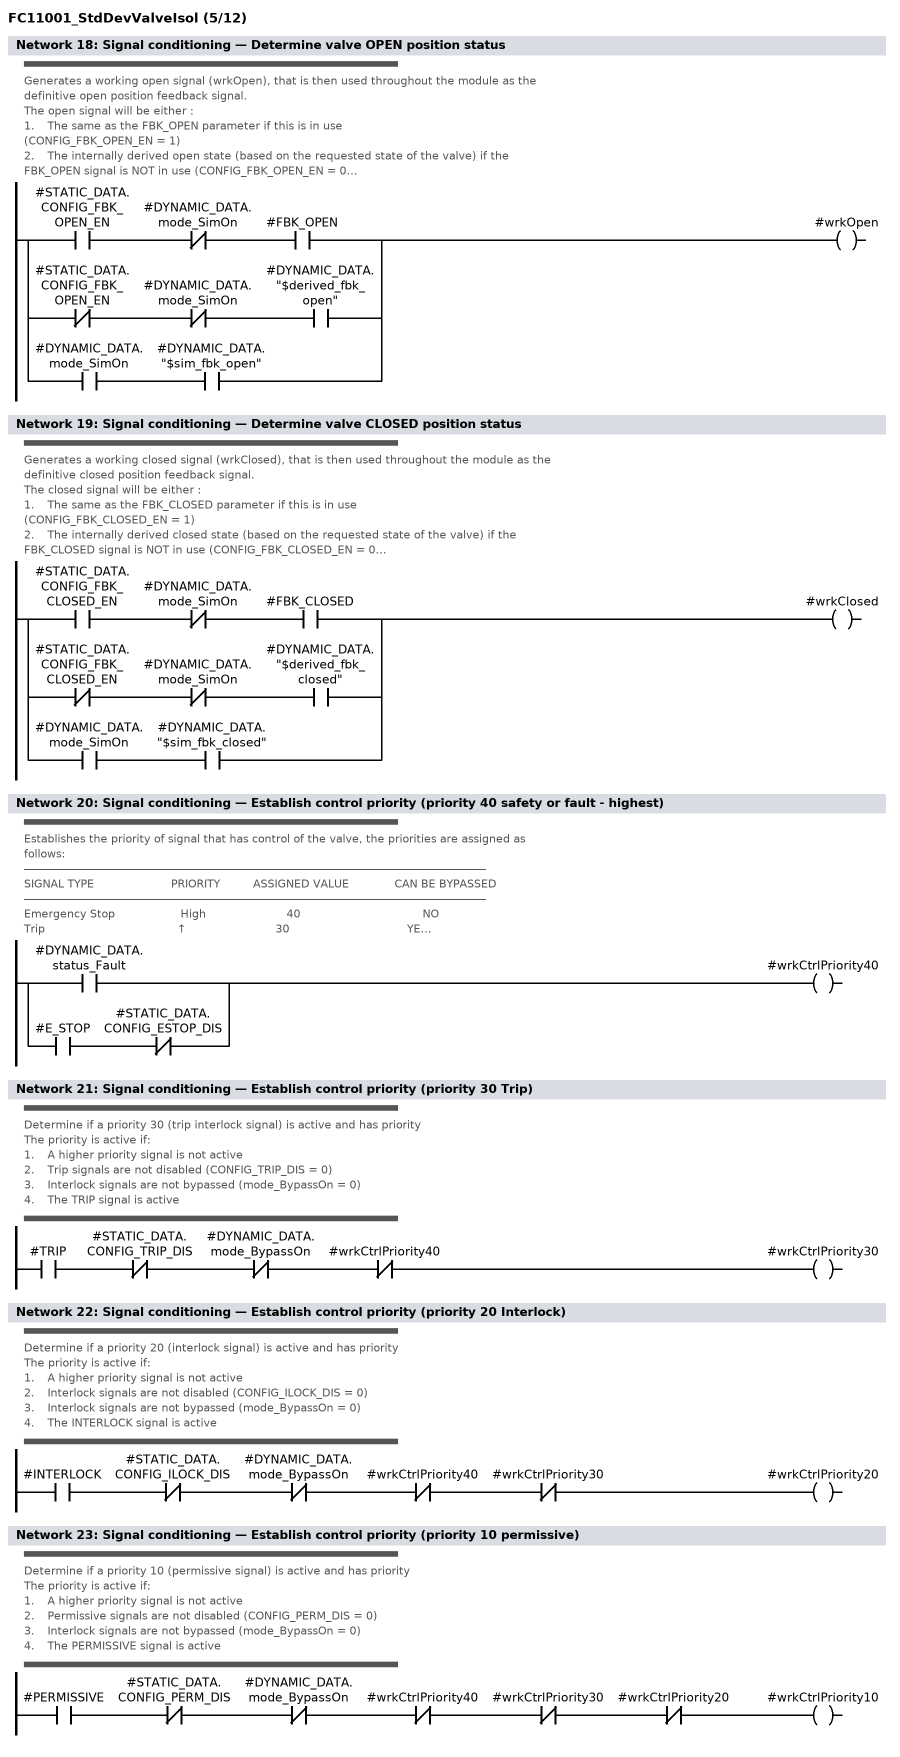
   RUNG wire#powerrail
      Contact( #STATIC_DATA.CONFIG_FBK_OPEN_EN )
      I_Contact( #DYNAMIC_DATA.mode_SimOn )
      Contact( #FBK_OPEN )
      wire#w1
      Coil( #wrkOpen )
   END_RUNG
   RUNG wire#powerrail
      I_Contact( #STATIC_DATA.CONFIG_FBK_OPEN_EN )
      I_Contact( #DYNAMIC_DATA.mode_SimOn )
      Contact( #DYNAMIC_DATA."$derived_fbk_open" )
   END_RUNG wire#w1
   RUNG wire#powerrail
      Contact( #DYNAMIC_DATA.mode_SimOn )
      Contact( #DYNAMIC_DATA."$sim_fbk_open" )
   END_RUNG wire#w1
   // the same network as SCL:
   #wrkOpen := (#STATIC_DATA.CONFIG_FBK_OPEN_EN AND NOT #DYNAMIC_DATA.mode_SimOn AND #FBK_OPEN) OR (NOT #STATIC_DATA.CONFIG_FBK_OPEN_EN AND NOT #DYNAMIC_DATA.mode_SimOn AND #DYNAMIC_DATA."$derived_fbk_open") OR (#DYNAMIC_DATA.mode_SimOn AND #DYNAMIC_DATA."$sim_fbk_open");
END_REGION

REGION Network 19: Signal conditioning — Determine valve CLOSED position status
   // ▀▀▀▀▀▀▀▀▀▀▀▀▀▀▀▀▀▀▀▀▀▀▀▀▀▀▀▀▀▀▀▀▀▀▀▀▀▀▀▀▀▀▀▀
   // Generates a working closed signal (wrkClosed), that is then used throughout the module as the 
   // definitive closed position feedback signal.
   // 
   // The closed signal will be either :
   // 
   //    1.  The same as the FBK_CLOSED parameter if this is in use 
   //      (CONFIG_FBK_CLOSED_EN = 1)
   // 
   //    2.  The internally derived closed state (based on the requested state of the valve) if the 
   //      FBK_CLOSED signal is NOT in use (CONFIG_FBK_CLOSED_EN = 0)
   // 
   //    3.  The simulated state of the valve if simulation mode is active (mode_SimOn = 1)
   // 
   // If an actual closed position signal is provided to the module via the FBK_CLOSED parameter 
   // (i.e. if CONFIG_FBK_CLOSED_EN = 1) then wrkClosed is set to match the FBK_CLOSED signal 
   // wrkClosed = FBK_CLOSED).
   // 
   // If a derived closed signal is to be used (i.e. if CONFIG_FBK_CLOSED_EN = 0), then wrkClosed is 
   // set to match the internally derived $derived_fbk_closed signal 
   // (wrkClosed = $derived_fbk_closed). $derived_fbk_closed is based on the requested state of 
   // the valve.
   // 
   // Finally, if simulation mode is active (mode_SimOn = 1), then wrkClosed is set to match the 
   // internal simulation signal $sim_fbk_closed signal (wrkClosed = $sim_fbk_closed). 
   // ▄▄▄▄▄▄▄▄▄▄▄▄▄▄▄▄▄▄▄▄▄▄▄▄▄▄▄▄▄▄▄▄▄▄▄▄▄▄▄▄▄▄▄▄
   RUNG wire#powerrail
      Contact( #STATIC_DATA.CONFIG_FBK_CLOSED_EN )
      I_Contact( #DYNAMIC_DATA.mode_SimOn )
      Contact( #FBK_CLOSED )
      wire#w1
      Coil( #wrkClosed )
   END_RUNG
   RUNG wire#powerrail
      I_Contact( #STATIC_DATA.CONFIG_FBK_CLOSED_EN )
      I_Contact( #DYNAMIC_DATA.mode_SimOn )
      Contact( #DYNAMIC_DATA."$derived_fbk_closed" )
   END_RUNG wire#w1
   RUNG wire#powerrail
      Contact( #DYNAMIC_DATA.mode_SimOn )
      Contact( #DYNAMIC_DATA."$sim_fbk_closed" )
   END_RUNG wire#w1
   // the same network as SCL:
   #wrkClosed := (#STATIC_DATA.CONFIG_FBK_CLOSED_EN AND NOT #DYNAMIC_DATA.mode_SimOn AND #FBK_CLOSED) OR (NOT #STATIC_DATA.CONFIG_FBK_CLOSED_EN AND NOT #DYNAMIC_DATA.mode_SimOn AND #DYNAMIC_DATA."$derived_fbk_closed") OR (#DYNAMIC_DATA.mode_SimOn AND #DYNAMIC_DATA."$sim_fbk_closed");
END_REGION

REGION Network 20: Signal conditioning — Establish control priority (priority 40 safety or fault - highest)
   // ▀▀▀▀▀▀▀▀▀▀▀▀▀▀▀▀▀▀▀▀▀▀▀▀▀▀▀▀▀▀▀▀▀▀▀▀▀▀▀▀▀▀▀▀
   // Establishes the priority of signal that has control of the valve, the priorities are assigned as 
   // follows:
   // 
   //  ――――――――――――――――――――――――――――――――――――――――――
   //  SIGNAL TYPE       PRIORITY   ASSIGNED VALUE       CAN BE BYPASSED
   //  ――――――――――――――――――――――――――――――――――――――――――
   //  Emergency Stop        High        40                NO
   //  Trip            ↑           30             YES
   //  Interlock            ↑           20             YES
   //  Permissive          ↑           10             YES
   //  Auto/manual control    Low         00                NO
   //  ――――――――――――――――――――――――――――――――――――――――――
   //  High priority signal take precedence over lower priority signals.
   // 
   // Determine a priority 40 (valve safety (or fault) condition is active)
   // 
   // The priority is active if:
   // 
   //    1.  The valve is in a fault condition (status_Fault = 1)
   // 
   //   OR both the following are true
   // 
   //    1.  Safety signals are not disabled (CONFIG_ESTOP_DIS = 0)
   // 
   //    2.  The E_STOP signal is active
   // ▄▄▄▄▄▄▄▄▄▄▄▄▄▄▄▄▄▄▄▄▄▄▄▄▄▄▄▄▄▄▄▄▄▄▄▄▄▄▄▄▄▄▄▄
   RUNG wire#powerrail
      Contact( #DYNAMIC_DATA.status_Fault )
      wire#w1
      Coil( #wrkCtrlPriority40 )
   END_RUNG
   RUNG wire#powerrail
      Contact( #E_STOP )
      I_Contact( #STATIC_DATA.CONFIG_ESTOP_DIS )
   END_RUNG wire#w1
   // the same network as SCL:
   #wrkCtrlPriority40 := #DYNAMIC_DATA.status_Fault OR (#E_STOP AND NOT #STATIC_DATA.CONFIG_ESTOP_DIS);
END_REGION

REGION Network 21: Signal conditioning — Establish control priority (priority 30 Trip)
   // ▀▀▀▀▀▀▀▀▀▀▀▀▀▀▀▀▀▀▀▀▀▀▀▀▀▀▀▀▀▀▀▀▀▀▀▀▀▀▀▀▀▀▀▀
   // Determine if a priority 30 (trip interlock signal) is active and has priority
   // 
   // The priority is active if:
   // 
   //    1.  A higher priority signal is not active
   // 
   //    2.  Trip signals are not disabled (CONFIG_TRIP_DIS = 0)
   // 
   //    3.  Interlock signals are not bypassed (mode_BypassOn = 0)
   // 
   //    4.  The TRIP signal is active
   // ▄▄▄▄▄▄▄▄▄▄▄▄▄▄▄▄▄▄▄▄▄▄▄▄▄▄▄▄▄▄▄▄▄▄▄▄▄▄▄▄▄▄▄▄
   RUNG wire#powerrail
      Contact( #TRIP )
      I_Contact( #STATIC_DATA.CONFIG_TRIP_DIS )
      I_Contact( #DYNAMIC_DATA.mode_BypassOn )
      I_Contact( #wrkCtrlPriority40 )
      Coil( #wrkCtrlPriority30 )
   END_RUNG
   // the same network as SCL:
   #wrkCtrlPriority30 := #TRIP AND NOT #STATIC_DATA.CONFIG_TRIP_DIS AND NOT #DYNAMIC_DATA.mode_BypassOn AND NOT #wrkCtrlPriority40;
END_REGION

REGION Network 22: Signal conditioning — Establish control priority (priority 20 Interlock)
   // ▀▀▀▀▀▀▀▀▀▀▀▀▀▀▀▀▀▀▀▀▀▀▀▀▀▀▀▀▀▀▀▀▀▀▀▀▀▀▀▀▀▀▀▀
   // Determine if a priority 20 (interlock signal) is active and has priority
   // 
   // The priority is active if:
   // 
   //    1.  A higher priority signal is not active
   // 
   //    2.  Interlock signals are not disabled (CONFIG_ILOCK_DIS = 0)
   // 
   //    3.  Interlock signals are not bypassed (mode_BypassOn = 0)
   // 
   //    4.  The INTERLOCK signal is active
   // ▄▄▄▄▄▄▄▄▄▄▄▄▄▄▄▄▄▄▄▄▄▄▄▄▄▄▄▄▄▄▄▄▄▄▄▄▄▄▄▄▄▄▄▄
   RUNG wire#powerrail
      Contact( #INTERLOCK )
      I_Contact( #STATIC_DATA.CONFIG_ILOCK_DIS )
      I_Contact( #DYNAMIC_DATA.mode_BypassOn )
      I_Contact( #wrkCtrlPriority40 )
      I_Contact( #wrkCtrlPriority30 )
      Coil( #wrkCtrlPriority20 )
   END_RUNG
   // the same network as SCL:
   #wrkCtrlPriority20 := #INTERLOCK AND NOT #STATIC_DATA.CONFIG_ILOCK_DIS AND NOT #DYNAMIC_DATA.mode_BypassOn AND NOT #wrkCtrlPriority40 AND NOT #wrkCtrlPriority30;
END_REGION

REGION Network 23: Signal conditioning — Establish control priority (priority 10 permissive)
   // ▀▀▀▀▀▀▀▀▀▀▀▀▀▀▀▀▀▀▀▀▀▀▀▀▀▀▀▀▀▀▀▀▀▀▀▀▀▀▀▀▀▀▀▀
   // Determine if a priority 10 (permissive signal) is active and has priority
   // 
   // The priority is active if:
   // 
   //    1.  A higher priority signal is not active
   // 
   //    2.  Permissive signals are not disabled (CONFIG_PERM_DIS = 0)
   // 
   //    3.  Interlock signals are not bypassed (mode_BypassOn = 0)
   // 
   //    4.  The PERMISSIVE signal is active
   // ▄▄▄▄▄▄▄▄▄▄▄▄▄▄▄▄▄▄▄▄▄▄▄▄▄▄▄▄▄▄▄▄▄▄▄▄▄▄▄▄▄▄▄▄
   RUNG wire#powerrail
      Contact( #PERMISSIVE )
      I_Contact( #STATIC_DATA.CONFIG_PERM_DIS )
      I_Contact( #DYNAMIC_DATA.mode_BypassOn )
      I_Contact( #wrkCtrlPriority40 )
      I_Contact( #wrkCtrlPriority30 )
      I_Contact( #wrkCtrlPriority20 )
      Coil( #wrkCtrlPriority10 )
   END_RUNG
   // the same network as SCL:
   #wrkCtrlPriority10 := #PERMISSIVE AND NOT #STATIC_DATA.CONFIG_PERM_DIS AND NOT #DYNAMIC_DATA.mode_BypassOn AND NOT #wrkCtrlPriority40 AND NOT #wrkCtrlPriority30 AND NOT #wrkCtrlPriority20;
END_REGION

REGION Network 24: Signal conditioning — Establish control priority (priority 00 auto/manual - lowest)
   // ▀▀▀▀▀▀▀▀▀▀▀▀▀▀▀▀▀▀▀▀▀▀▀▀▀▀▀▀▀▀▀▀▀▀▀▀▀▀▀▀▀▀▀▀
   // Determine if a priority 00 (automatic or manual control) is active and has priority
   // 
   // The priority is active if:
   // 
   //    1.  A higher priority signal is not active
   // ▄▄▄▄▄▄▄▄▄▄▄▄▄▄▄▄▄▄▄▄▄▄▄▄▄▄▄▄▄▄▄▄▄▄▄▄▄▄▄▄▄▄▄▄
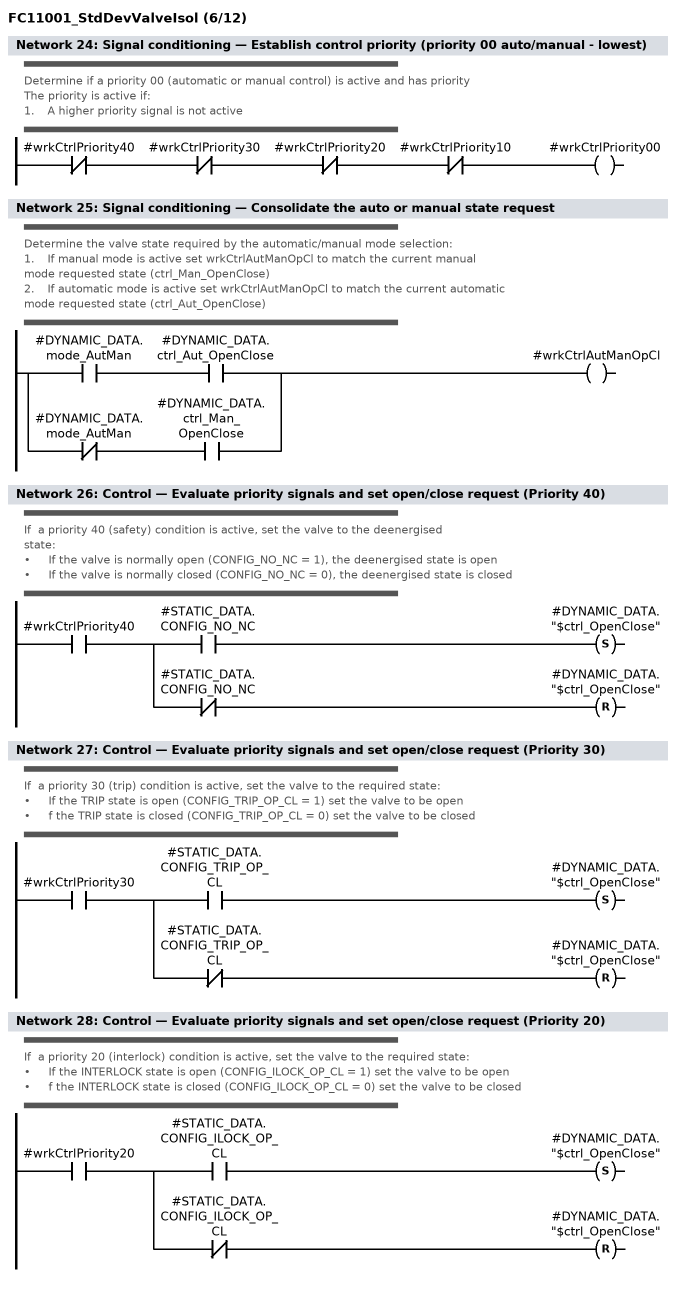
   RUNG wire#powerrail
      I_Contact( #wrkCtrlPriority40 )
      I_Contact( #wrkCtrlPriority30 )
      I_Contact( #wrkCtrlPriority20 )
      I_Contact( #wrkCtrlPriority10 )
      Coil( #wrkCtrlPriority00 )
   END_RUNG
   // the same network as SCL:
   #wrkCtrlPriority00 := NOT #wrkCtrlPriority40 AND NOT #wrkCtrlPriority30 AND NOT #wrkCtrlPriority20 AND NOT #wrkCtrlPriority10;
END_REGION

REGION Network 25: Signal conditioning — Consolidate the auto or manual state request
   // ▀▀▀▀▀▀▀▀▀▀▀▀▀▀▀▀▀▀▀▀▀▀▀▀▀▀▀▀▀▀▀▀▀▀▀▀▀▀▀▀▀▀▀▀
   // Determine the valve state required by the automatic/manual mode selection:
   // 
   //    1.  If manual mode is active set wrkCtrlAutManOpCl to match the current manual 
   //      mode requested state (ctrl_Man_OpenClose)
   // 
   //    2.  If automatic mode is active set wrkCtrlAutManOpCl to match the current automatic 
   //      mode requested state (ctrl_Aut_OpenClose)
   // ▄▄▄▄▄▄▄▄▄▄▄▄▄▄▄▄▄▄▄▄▄▄▄▄▄▄▄▄▄▄▄▄▄▄▄▄▄▄▄▄▄▄▄▄
   RUNG wire#powerrail
      Contact( #DYNAMIC_DATA.mode_AutMan )
      Contact( #DYNAMIC_DATA.ctrl_Aut_OpenClose )
      wire#w1
      Coil( #wrkCtrlAutManOpCl )
   END_RUNG
   RUNG wire#powerrail
      I_Contact( #DYNAMIC_DATA.mode_AutMan )
      Contact( #DYNAMIC_DATA.ctrl_Man_OpenClose )
   END_RUNG wire#w1
   // the same network as SCL:
   #wrkCtrlAutManOpCl := (#DYNAMIC_DATA.mode_AutMan AND #DYNAMIC_DATA.ctrl_Aut_OpenClose) OR (NOT #DYNAMIC_DATA.mode_AutMan AND #DYNAMIC_DATA.ctrl_Man_OpenClose);
END_REGION

REGION Network 26: Control — Evaluate priority signals and set open/close request (Priority 40)
   // ▀▀▀▀▀▀▀▀▀▀▀▀▀▀▀▀▀▀▀▀▀▀▀▀▀▀▀▀▀▀▀▀▀▀▀▀▀▀▀▀▀▀▀▀
   // If  a priority 40 (safety) condition is active, set the valve to the deenergised 
   // state:
   // 
   //    •   If the valve is normally open (CONFIG_NO_NC = 1), the deenergised state is open
   // 
   //    •   If the valve is normally closed (CONFIG_NO_NC = 0), the deenergised state is closed
   // ▄▄▄▄▄▄▄▄▄▄▄▄▄▄▄▄▄▄▄▄▄▄▄▄▄▄▄▄▄▄▄▄▄▄▄▄▄▄▄▄▄▄▄▄
   RUNG wire#powerrail
      Contact( #wrkCtrlPriority40 )
      wire#w1
      Contact( #STATIC_DATA.CONFIG_NO_NC )
      S_Coil( #DYNAMIC_DATA."$ctrl_OpenClose" )
   END_RUNG
   RUNG wire#w1
      I_Contact( #STATIC_DATA.CONFIG_NO_NC )
      R_Coil( #DYNAMIC_DATA."$ctrl_OpenClose" )
   END_RUNG
   // the same network as SCL:
   IF #wrkCtrlPriority40 AND #STATIC_DATA.CONFIG_NO_NC THEN #DYNAMIC_DATA."$ctrl_OpenClose" := TRUE; END_IF;
   IF #wrkCtrlPriority40 AND NOT #STATIC_DATA.CONFIG_NO_NC THEN
       #DYNAMIC_DATA."$ctrl_OpenClose" := FALSE;
   END_IF;
END_REGION

REGION Network 27: Control — Evaluate priority signals and set open/close request (Priority 30)
   // ▀▀▀▀▀▀▀▀▀▀▀▀▀▀▀▀▀▀▀▀▀▀▀▀▀▀▀▀▀▀▀▀▀▀▀▀▀▀▀▀▀▀▀▀
   // If  a priority 30 (trip) condition is active, set the valve to the required state:
   // 
   //    •   If the TRIP state is open (CONFIG_TRIP_OP_CL = 1) set the valve to be open
   // 
   //    •   f the TRIP state is closed (CONFIG_TRIP_OP_CL = 0) set the valve to be closed
   // ▄▄▄▄▄▄▄▄▄▄▄▄▄▄▄▄▄▄▄▄▄▄▄▄▄▄▄▄▄▄▄▄▄▄▄▄▄▄▄▄▄▄▄▄
   RUNG wire#powerrail
      Contact( #wrkCtrlPriority30 )
      wire#w1
      Contact( #STATIC_DATA.CONFIG_TRIP_OP_CL )
      S_Coil( #DYNAMIC_DATA."$ctrl_OpenClose" )
   END_RUNG
   RUNG wire#w1
      I_Contact( #STATIC_DATA.CONFIG_TRIP_OP_CL )
      R_Coil( #DYNAMIC_DATA."$ctrl_OpenClose" )
   END_RUNG
   // the same network as SCL:
   IF #wrkCtrlPriority30 AND #STATIC_DATA.CONFIG_TRIP_OP_CL THEN
       #DYNAMIC_DATA."$ctrl_OpenClose" := TRUE;
   END_IF;
   IF #wrkCtrlPriority30 AND NOT #STATIC_DATA.CONFIG_TRIP_OP_CL THEN
       #DYNAMIC_DATA."$ctrl_OpenClose" := FALSE;
   END_IF;
END_REGION

REGION Network 28: Control — Evaluate priority signals and set open/close request (Priority 20)
   // ▀▀▀▀▀▀▀▀▀▀▀▀▀▀▀▀▀▀▀▀▀▀▀▀▀▀▀▀▀▀▀▀▀▀▀▀▀▀▀▀▀▀▀▀
   // If  a priority 20 (interlock) condition is active, set the valve to the required state:
   // 
   //    •   If the INTERLOCK state is open (CONFIG_ILOCK_OP_CL = 1) set the valve to be open
   // 
   //    •   f the INTERLOCK state is closed (CONFIG_ILOCK_OP_CL = 0) set the valve to be closed
   // ▄▄▄▄▄▄▄▄▄▄▄▄▄▄▄▄▄▄▄▄▄▄▄▄▄▄▄▄▄▄▄▄▄▄▄▄▄▄▄▄▄▄▄▄
   RUNG wire#powerrail
      Contact( #wrkCtrlPriority20 )
      wire#w1
      Contact( #STATIC_DATA.CONFIG_ILOCK_OP_CL )
      S_Coil( #DYNAMIC_DATA."$ctrl_OpenClose" )
   END_RUNG
   RUNG wire#w1
      I_Contact( #STATIC_DATA.CONFIG_ILOCK_OP_CL )
      R_Coil( #DYNAMIC_DATA."$ctrl_OpenClose" )
   END_RUNG
   // the same network as SCL:
   IF #wrkCtrlPriority20 AND #STATIC_DATA.CONFIG_ILOCK_OP_CL THEN
       #DYNAMIC_DATA."$ctrl_OpenClose" := TRUE;
   END_IF;
   IF #wrkCtrlPriority20 AND NOT #STATIC_DATA.CONFIG_ILOCK_OP_CL THEN
       #DYNAMIC_DATA."$ctrl_OpenClose" := FALSE;
   END_IF;
END_REGION

REGION Network 29: Control — Evaluate priority signals and set open/close request (Priority 10)
   // ▀▀▀▀▀▀▀▀▀▀▀▀▀▀▀▀▀▀▀▀▀▀▀▀▀▀▀▀▀▀▀▀▀▀▀▀▀▀▀▀▀▀▀▀
   // If  a priority 10 (permissive) condition is active, set the valve to the required state:
   // 
   // 
   // PERMITTED STATE IS OPEN — CONDITIONS:
   // 
   //    •   If the Permitted state is open and Aut/Man request is for open, 
   //      set the valve to be open [Branch 1]
   // 
   //    •   If the Permitted state is open and Aut/Man request is for closed, and the current
   //      valve output matches this state (closed), set the valve to be closed (maintain the
   //      current state) [Branch 6]
   // 
   //    •   If the Permitted state is open and Aut/Man request is for closed, and the current
   //      valve output matches the open state, set the valve to be open (override the
   //      auto/man request [Branch 2]
   // 
   // PERMITTED STATE IS CLOSED — CONDITIONS:
   // 
   //    •   If the Permitted state is closed and Aut/Man request is for closed,
   //      set the valve to be  closed [Branch 4]
   // 
   //    •   If the Permitted state is closed and Aut/Man request is for open, and the current
   //      valve output matches this state (open), set the valve to be open (maintain the
   //      current state) [Branch 3]
   // 
   //    •   If the Permitted state is closed and Aut/Man request is for open, and the current
   //      valve output matches the closed state, set the valve to be closed (override the
   //      auto/man request [Branch 5]
   // ▄▄▄▄▄▄▄▄▄▄▄▄▄▄▄▄▄▄▄▄▄▄▄▄▄▄▄▄▄▄▄▄▄▄▄▄▄▄▄▄▄▄▄▄
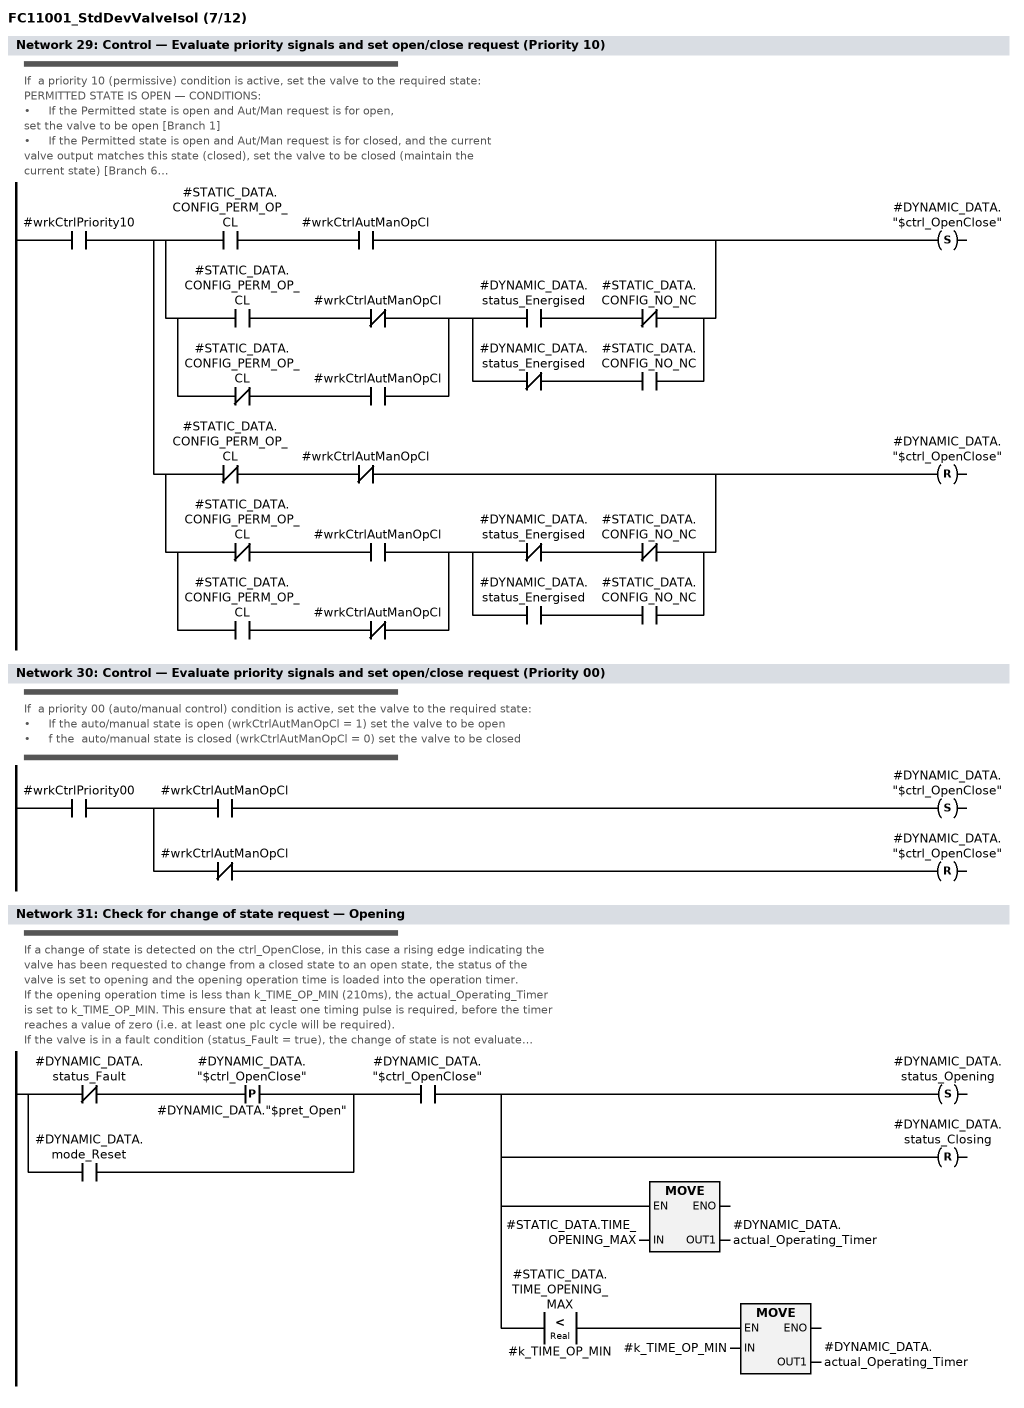
   RUNG wire#powerrail
      Contact( #wrkCtrlPriority10 )
      wire#w1
      Contact( #STATIC_DATA.CONFIG_PERM_OP_CL )
      Contact( #wrkCtrlAutManOpCl )
      wire#w2
      S_Coil( #DYNAMIC_DATA."$ctrl_OpenClose" )
   END_RUNG
   RUNG wire#w1
      Contact( #STATIC_DATA.CONFIG_PERM_OP_CL )
      I_Contact( #wrkCtrlAutManOpCl )
      wire#w3
      Contact( #DYNAMIC_DATA.status_Energised )
      I_Contact( #STATIC_DATA.CONFIG_NO_NC )
   END_RUNG wire#w2
   RUNG wire#w1
      I_Contact( #STATIC_DATA.CONFIG_PERM_OP_CL )
      Contact( #wrkCtrlAutManOpCl )
   END_RUNG wire#w3
   RUNG wire#w3
      I_Contact( #DYNAMIC_DATA.status_Energised )
      Contact( #STATIC_DATA.CONFIG_NO_NC )
   END_RUNG wire#w2
   RUNG wire#w1
      I_Contact( #STATIC_DATA.CONFIG_PERM_OP_CL )
      I_Contact( #wrkCtrlAutManOpCl )
      wire#w4
      R_Coil( #DYNAMIC_DATA."$ctrl_OpenClose" )
   END_RUNG
   RUNG wire#w1
      I_Contact( #STATIC_DATA.CONFIG_PERM_OP_CL )
      Contact( #wrkCtrlAutManOpCl )
      wire#w5
      I_Contact( #DYNAMIC_DATA.status_Energised )
      I_Contact( #STATIC_DATA.CONFIG_NO_NC )
   END_RUNG wire#w4
   RUNG wire#w1
      Contact( #STATIC_DATA.CONFIG_PERM_OP_CL )
      I_Contact( #wrkCtrlAutManOpCl )
   END_RUNG wire#w5
   RUNG wire#w5
      Contact( #DYNAMIC_DATA.status_Energised )
      Contact( #STATIC_DATA.CONFIG_NO_NC )
   END_RUNG wire#w4
   // the same network as SCL:
   IF #wrkCtrlPriority10 AND ((#STATIC_DATA.CONFIG_PERM_OP_CL AND #wrkCtrlAutManOpCl) OR (((#STATIC_DATA.CONFIG_PERM_OP_CL AND NOT #wrkCtrlAutManOpCl) OR (NOT #STATIC_DATA.CONFIG_PERM_OP_CL AND #wrkCtrlAutManOpCl)) AND ((#DYNAMIC_DATA.status_Energised AND NOT #STATIC_DATA.CONFIG_NO_NC) OR (NOT #DYNAMIC_DATA.status_Energised AND #STATIC_DATA.CONFIG_NO_NC)))) THEN
       #DYNAMIC_DATA."$ctrl_OpenClose" := TRUE;
   END_IF;
   IF #wrkCtrlPriority10 AND ((NOT #STATIC_DATA.CONFIG_PERM_OP_CL AND NOT #wrkCtrlAutManOpCl) OR (((NOT #STATIC_DATA.CONFIG_PERM_OP_CL AND #wrkCtrlAutManOpCl) OR (#STATIC_DATA.CONFIG_PERM_OP_CL AND NOT #wrkCtrlAutManOpCl)) AND ((NOT #DYNAMIC_DATA.status_Energised AND NOT #STATIC_DATA.CONFIG_NO_NC) OR (#DYNAMIC_DATA.status_Energised AND #STATIC_DATA.CONFIG_NO_NC)))) THEN
       #DYNAMIC_DATA."$ctrl_OpenClose" := FALSE;
   END_IF;
END_REGION

REGION Network 30: Control — Evaluate priority signals and set open/close request (Priority 00)
   // ▀▀▀▀▀▀▀▀▀▀▀▀▀▀▀▀▀▀▀▀▀▀▀▀▀▀▀▀▀▀▀▀▀▀▀▀▀▀▀▀▀▀▀▀
   // If  a priority 00 (auto/manual control) condition is active, set the valve to the required state:
   // 
   //    •   If the auto/manual state is open (wrkCtrlAutManOpCl = 1) set the valve to be open
   // 
   //    •   f the  auto/manual state is closed (wrkCtrlAutManOpCl = 0) set the valve to be closed
   // ▄▄▄▄▄▄▄▄▄▄▄▄▄▄▄▄▄▄▄▄▄▄▄▄▄▄▄▄▄▄▄▄▄▄▄▄▄▄▄▄▄▄▄▄
   RUNG wire#powerrail
      Contact( #wrkCtrlPriority00 )
      wire#w1
      Contact( #wrkCtrlAutManOpCl )
      S_Coil( #DYNAMIC_DATA."$ctrl_OpenClose" )
   END_RUNG
   RUNG wire#w1
      I_Contact( #wrkCtrlAutManOpCl )
      R_Coil( #DYNAMIC_DATA."$ctrl_OpenClose" )
   END_RUNG
   // the same network as SCL:
   IF #wrkCtrlPriority00 AND #wrkCtrlAutManOpCl THEN #DYNAMIC_DATA."$ctrl_OpenClose" := TRUE; END_IF;
   IF #wrkCtrlPriority00 AND NOT #wrkCtrlAutManOpCl THEN #DYNAMIC_DATA."$ctrl_OpenClose" := FALSE; END_IF;
END_REGION

REGION Network 31: Check for change of state request — Opening
   // ▀▀▀▀▀▀▀▀▀▀▀▀▀▀▀▀▀▀▀▀▀▀▀▀▀▀▀▀▀▀▀▀▀▀▀▀▀▀▀▀▀▀▀▀
   // If a change of state is detected on the ctrl_OpenClose, in this case a rising edge indicating the
   // valve has been requested to change from a closed state to an open state, the status of the
   // valve is set to opening and the opening operation time is loaded into the operation timer.
   // 
   // If the opening operation time is less than k_TIME_OP_MIN (210ms), the actual_Operating_Timer 
   // is set to k_TIME_OP_MIN. This ensure that at least one timing pulse is required, before the timer 
   // reaches a value of zero (i.e. at least one plc cycle will be required).
   // 
   // If the valve is in a fault condition (status_Fault = true), the change of state is not evaluated
   // until the fault condition has cleared
   // 
   // Note: the timer is also triggered if the Reset signal is received and the valve is requested open.
   // ▄▄▄▄▄▄▄▄▄▄▄▄▄▄▄▄▄▄▄▄▄▄▄▄▄▄▄▄▄▄▄▄▄▄▄▄▄▄▄▄▄▄▄▄
   RUNG wire#powerrail
      I_Contact( #DYNAMIC_DATA.status_Fault )
      P_Contact(operand := #DYNAMIC_DATA."$ctrl_OpenClose", bit := #DYNAMIC_DATA."$pret_Open")
      wire#w1
      Contact( #DYNAMIC_DATA."$ctrl_OpenClose" )
      wire#w2
      S_Coil( #DYNAMIC_DATA.status_Opening )
   END_RUNG
   RUNG wire#powerrail
      Contact( #DYNAMIC_DATA.mode_Reset )
   END_RUNG wire#w1
   RUNG wire#w2
      R_Coil( #DYNAMIC_DATA.status_Closing )
   END_RUNG
   RUNG wire#w2
      Move(in := #STATIC_DATA.TIME_OPENING_MAX, out1 => #DYNAMIC_DATA.actual_Operating_Timer)
   END_RUNG
   RUNG wire#w2
      { S7_Templates := "SrcType := Real" } LT_Contact(in1 := #STATIC_DATA.TIME_OPENING_MAX, in2 := #k_TIME_OP_MIN)
      Move(in := #k_TIME_OP_MIN, out1 => #DYNAMIC_DATA.actual_Operating_Timer)
   END_RUNG
   // the same network as SCL:
   #_w1 := NOT #DYNAMIC_DATA.status_Fault AND #DYNAMIC_DATA."$ctrl_OpenClose" AND NOT #DYNAMIC_DATA."$pret_Open";   // rising edge of #DYNAMIC_DATA."$ctrl_OpenClose"
   #DYNAMIC_DATA."$pret_Open" := #DYNAMIC_DATA."$ctrl_OpenClose";
   #_w2 := (#_w1 OR #DYNAMIC_DATA.mode_Reset) AND #DYNAMIC_DATA."$ctrl_OpenClose";
   IF #_w2 THEN
       #DYNAMIC_DATA.status_Opening := TRUE;
       #DYNAMIC_DATA.status_Closing := FALSE;
       #DYNAMIC_DATA.actual_Operating_Timer := #STATIC_DATA.TIME_OPENING_MAX;
   END_IF;
   IF #_w2 AND (#STATIC_DATA.TIME_OPENING_MAX < #k_TIME_OP_MIN) THEN
       #DYNAMIC_DATA.actual_Operating_Timer := #k_TIME_OP_MIN;
   END_IF;
END_REGION

REGION Network 32: Check for change of state request — Closing
   // ▀▀▀▀▀▀▀▀▀▀▀▀▀▀▀▀▀▀▀▀▀▀▀▀▀▀▀▀▀▀▀▀▀▀▀▀▀▀▀▀▀▀▀▀
   // If a change of state is detected on the ctrl_OpenClose, in this case a falling edge indicating the
   // valve has been requested to change from an open state to a closed state, the status of the
   // valve is set to closing and the closing operation time is loaded into the operation timer.
   // 
   // If the closing operation time is less than k_TIME_OP_MIN (210ms), the actual_Operating_Timer 
   // is set to k_TIME_OP_MIN. This ensure that at least one timing pulse is required, before the timer 
   // reaches a value of zero (i.e. at least one plc cycle will be required).
   // 
   // If the valve is in a fault condition (status_Fault = true), the change of state is not evaluated
   // until the fault condition has cleared
   // 
   // Note: the timer is also triggered if the Reset signal is received and the valve is requested closed.
   // ▄▄▄▄▄▄▄▄▄▄▄▄▄▄▄▄▄▄▄▄▄▄▄▄▄▄▄▄▄▄▄▄▄▄▄▄▄▄▄▄▄▄▄▄
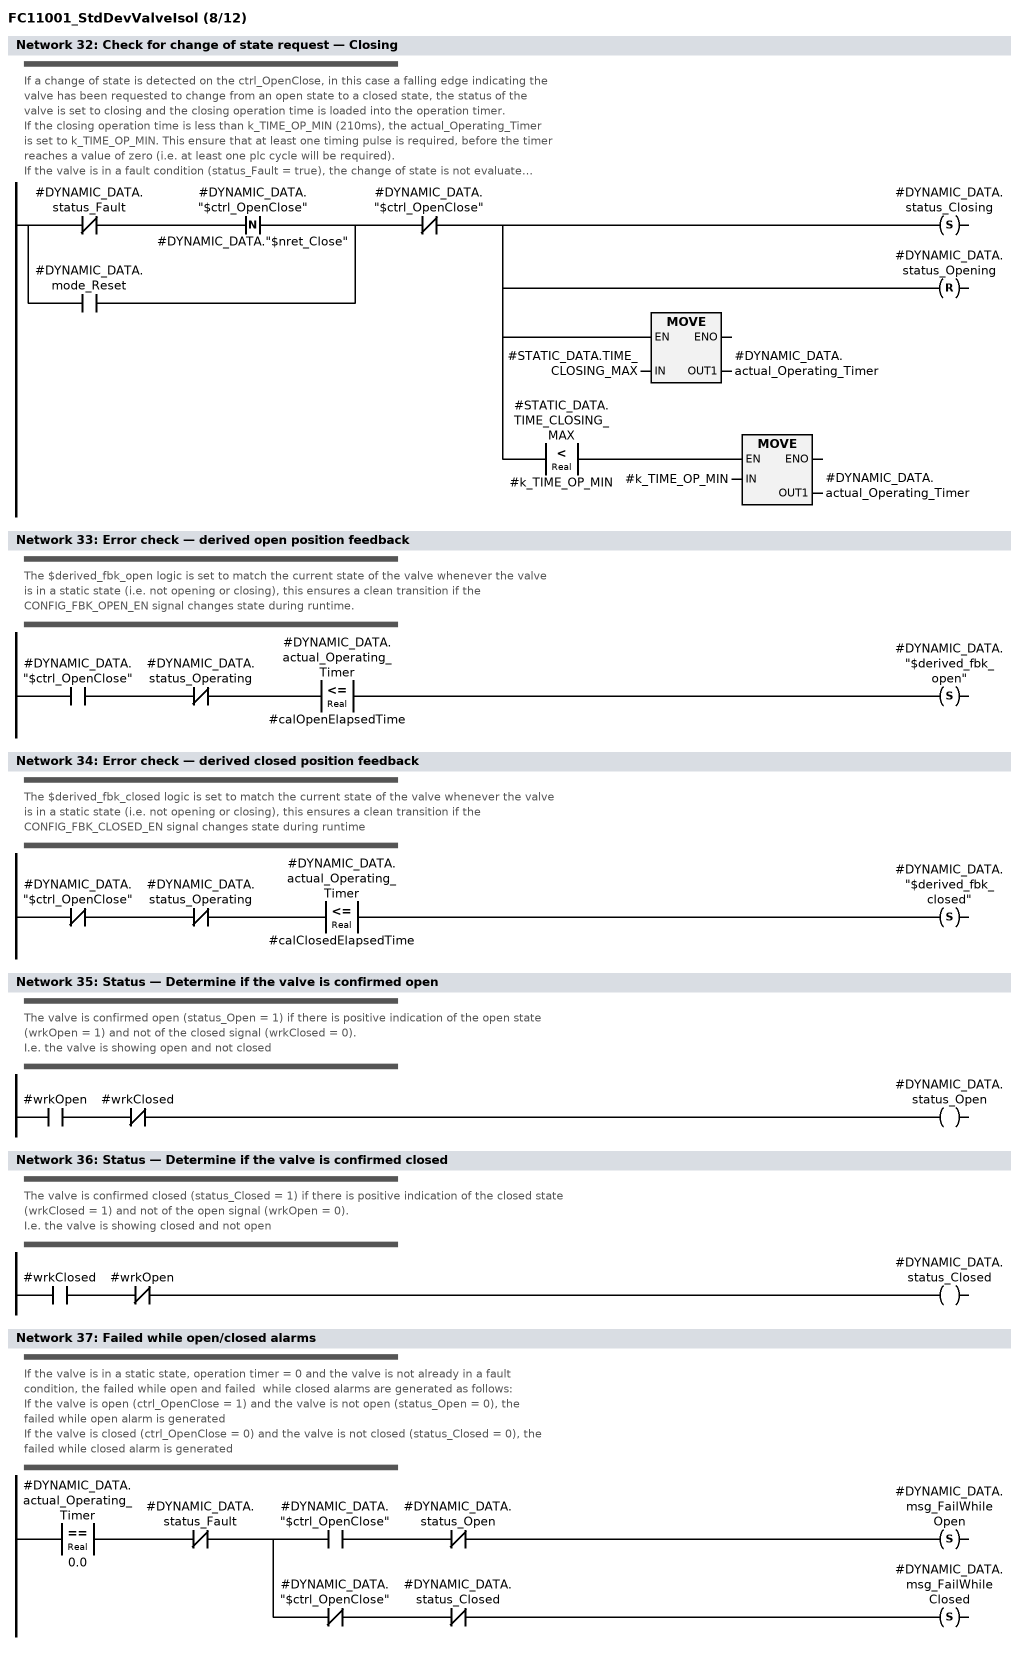
   RUNG wire#powerrail
      I_Contact( #DYNAMIC_DATA.status_Fault )
      N_Contact(operand := #DYNAMIC_DATA."$ctrl_OpenClose", bit := #DYNAMIC_DATA."$nret_Close")
      wire#w1
      I_Contact( #DYNAMIC_DATA."$ctrl_OpenClose" )
      wire#w2
      S_Coil( #DYNAMIC_DATA.status_Closing )
   END_RUNG
   RUNG wire#powerrail
      Contact( #DYNAMIC_DATA.mode_Reset )
   END_RUNG wire#w1
   RUNG wire#w2
      R_Coil( #DYNAMIC_DATA.status_Opening )
   END_RUNG
   RUNG wire#w2
      Move(in := #STATIC_DATA.TIME_CLOSING_MAX, out1 => #DYNAMIC_DATA.actual_Operating_Timer)
   END_RUNG
   RUNG wire#w2
      { S7_Templates := "SrcType := Real" } LT_Contact(in1 := #STATIC_DATA.TIME_CLOSING_MAX, in2 := #k_TIME_OP_MIN)
      Move(in := #k_TIME_OP_MIN, out1 => #DYNAMIC_DATA.actual_Operating_Timer)
   END_RUNG
   // the same network as SCL:
   #_w1 := NOT #DYNAMIC_DATA.status_Fault AND NOT #DYNAMIC_DATA."$ctrl_OpenClose" AND #DYNAMIC_DATA."$nret_Close";   // falling edge of #DYNAMIC_DATA."$ctrl_OpenClose"
   #DYNAMIC_DATA."$nret_Close" := #DYNAMIC_DATA."$ctrl_OpenClose";
   #_w2 := (#_w1 OR #DYNAMIC_DATA.mode_Reset) AND NOT #DYNAMIC_DATA."$ctrl_OpenClose";
   IF #_w2 THEN
       #DYNAMIC_DATA.status_Closing := TRUE;
       #DYNAMIC_DATA.status_Opening := FALSE;
       #DYNAMIC_DATA.actual_Operating_Timer := #STATIC_DATA.TIME_CLOSING_MAX;
   END_IF;
   IF #_w2 AND (#STATIC_DATA.TIME_CLOSING_MAX < #k_TIME_OP_MIN) THEN
       #DYNAMIC_DATA.actual_Operating_Timer := #k_TIME_OP_MIN;
   END_IF;
END_REGION

REGION Network 33: Error check — derived open position feedback
   // ▀▀▀▀▀▀▀▀▀▀▀▀▀▀▀▀▀▀▀▀▀▀▀▀▀▀▀▀▀▀▀▀▀▀▀▀▀▀▀▀▀▀▀▀
   // The $derived_fbk_open logic is set to match the current state of the valve whenever the valve
   // is in a static state (i.e. not opening or closing), this ensures a clean transition if the 
   // CONFIG_FBK_OPEN_EN signal changes state during runtime.
   // ▄▄▄▄▄▄▄▄▄▄▄▄▄▄▄▄▄▄▄▄▄▄▄▄▄▄▄▄▄▄▄▄▄▄▄▄▄▄▄▄▄▄▄▄
   RUNG wire#powerrail
      Contact( #DYNAMIC_DATA."$ctrl_OpenClose" )
      I_Contact( #DYNAMIC_DATA.status_Operating )
      { S7_Templates := "SrcType := Real" } LE_Contact(in1 := #DYNAMIC_DATA.actual_Operating_Timer, in2 := #calOpenElapsedTime)
      S_Coil( #DYNAMIC_DATA."$derived_fbk_open" )
   END_RUNG
   // the same network as SCL:
   IF #DYNAMIC_DATA."$ctrl_OpenClose" AND NOT #DYNAMIC_DATA.status_Operating AND (#DYNAMIC_DATA.actual_Operating_Timer <= #calOpenElapsedTime) THEN
       #DYNAMIC_DATA."$derived_fbk_open" := TRUE;
   END_IF;
END_REGION

REGION Network 34: Error check — derived closed position feedback
   // ▀▀▀▀▀▀▀▀▀▀▀▀▀▀▀▀▀▀▀▀▀▀▀▀▀▀▀▀▀▀▀▀▀▀▀▀▀▀▀▀▀▀▀▀
   // The $derived_fbk_closed logic is set to match the current state of the valve whenever the valve
   // is in a static state (i.e. not opening or closing), this ensures a clean transition if the 
   // CONFIG_FBK_CLOSED_EN signal changes state during runtime
   // ▄▄▄▄▄▄▄▄▄▄▄▄▄▄▄▄▄▄▄▄▄▄▄▄▄▄▄▄▄▄▄▄▄▄▄▄▄▄▄▄▄▄▄▄
   RUNG wire#powerrail
      I_Contact( #DYNAMIC_DATA."$ctrl_OpenClose" )
      I_Contact( #DYNAMIC_DATA.status_Operating )
      { S7_Templates := "SrcType := Real" } LE_Contact(in1 := #DYNAMIC_DATA.actual_Operating_Timer, in2 := #calClosedElapsedTime)
      S_Coil( #DYNAMIC_DATA."$derived_fbk_closed" )
   END_RUNG
   // the same network as SCL:
   IF NOT #DYNAMIC_DATA."$ctrl_OpenClose" AND NOT #DYNAMIC_DATA.status_Operating AND (#DYNAMIC_DATA.actual_Operating_Timer <= #calClosedElapsedTime) THEN
       #DYNAMIC_DATA."$derived_fbk_closed" := TRUE;
   END_IF;
END_REGION

REGION Network 35: Status — Determine if the valve is confirmed open
   // ▀▀▀▀▀▀▀▀▀▀▀▀▀▀▀▀▀▀▀▀▀▀▀▀▀▀▀▀▀▀▀▀▀▀▀▀▀▀▀▀▀▀▀▀
   // The valve is confirmed open (status_Open = 1) if there is positive indication of the open state 
   // (wrkOpen = 1) and not of the closed signal (wrkClosed = 0). 
   // 
   // I.e. the valve is showing open and not closed
   // ▄▄▄▄▄▄▄▄▄▄▄▄▄▄▄▄▄▄▄▄▄▄▄▄▄▄▄▄▄▄▄▄▄▄▄▄▄▄▄▄▄▄▄▄
   RUNG wire#powerrail
      Contact( #wrkOpen )
      I_Contact( #wrkClosed )
      Coil( #DYNAMIC_DATA.status_Open )
   END_RUNG
   // the same network as SCL:
   #DYNAMIC_DATA.status_Open := #wrkOpen AND NOT #wrkClosed;
END_REGION

REGION Network 36: Status — Determine if the valve is confirmed closed
   // ▀▀▀▀▀▀▀▀▀▀▀▀▀▀▀▀▀▀▀▀▀▀▀▀▀▀▀▀▀▀▀▀▀▀▀▀▀▀▀▀▀▀▀▀
   // The valve is confirmed closed (status_Closed = 1) if there is positive indication of the closed state 
   // (wrkClosed = 1) and not of the open signal (wrkOpen = 0). 
   // 
   // I.e. the valve is showing closed and not open
   // ▄▄▄▄▄▄▄▄▄▄▄▄▄▄▄▄▄▄▄▄▄▄▄▄▄▄▄▄▄▄▄▄▄▄▄▄▄▄▄▄▄▄▄▄
   RUNG wire#powerrail
      Contact( #wrkClosed )
      I_Contact( #wrkOpen )
      Coil( #DYNAMIC_DATA.status_Closed )
   END_RUNG
   // the same network as SCL:
   #DYNAMIC_DATA.status_Closed := #wrkClosed AND NOT #wrkOpen;
END_REGION

REGION Network 37: Failed while open/closed alarms
   // ▀▀▀▀▀▀▀▀▀▀▀▀▀▀▀▀▀▀▀▀▀▀▀▀▀▀▀▀▀▀▀▀▀▀▀▀▀▀▀▀▀▀▀▀
   // If the valve is in a static state, operation timer = 0 and the valve is not already in a fault
   // condition, the failed while open and failed  while closed alarms are generated as follows:
   // 
   // If the valve is open (ctrl_OpenClose = 1) and the valve is not open (status_Open = 0), the 
   // failed while open alarm is generated
   // 
   // If the valve is closed (ctrl_OpenClose = 0) and the valve is not closed (status_Closed = 0), the 
   // failed while closed alarm is generated
   // ▄▄▄▄▄▄▄▄▄▄▄▄▄▄▄▄▄▄▄▄▄▄▄▄▄▄▄▄▄▄▄▄▄▄▄▄▄▄▄▄▄▄▄▄
   RUNG wire#powerrail
      { S7_Templates := "SrcType := Real" } EQ_Contact(in1 := #DYNAMIC_DATA.actual_Operating_Timer, in2 := 0.0)
      I_Contact( #DYNAMIC_DATA.status_Fault )
      wire#w1
      Contact( #DYNAMIC_DATA."$ctrl_OpenClose" )
      I_Contact( #DYNAMIC_DATA.status_Open )
      S_Coil( #DYNAMIC_DATA.msg_FailWhileOpen )
   END_RUNG
   RUNG wire#w1
      I_Contact( #DYNAMIC_DATA."$ctrl_OpenClose" )
      I_Contact( #DYNAMIC_DATA.status_Closed )
      S_Coil( #DYNAMIC_DATA.msg_FailWhileClosed )
   END_RUNG
   // the same network as SCL:
   #_w1 := (#DYNAMIC_DATA.actual_Operating_Timer = 0.0) AND NOT #DYNAMIC_DATA.status_Fault;
   IF #_w1 AND #DYNAMIC_DATA."$ctrl_OpenClose" AND NOT #DYNAMIC_DATA.status_Open THEN
       #DYNAMIC_DATA.msg_FailWhileOpen := TRUE;
   END_IF;
   IF #_w1 AND NOT #DYNAMIC_DATA."$ctrl_OpenClose" AND NOT #DYNAMIC_DATA.status_Closed THEN
       #DYNAMIC_DATA.msg_FailWhileClosed := TRUE;
   END_IF;
END_REGION

REGION Network 38: Operation timer and Failed to open/close alarms
   // ▀▀▀▀▀▀▀▀▀▀▀▀▀▀▀▀▀▀▀▀▀▀▀▀▀▀▀▀▀▀▀▀▀▀▀▀▀▀▀▀▀▀▀▀
   // If the valve is opening or closing, decrement the current operation timer value on each 200ms
   // pulse.
   // 
   // If the timer reaches zero, and the valve is opening, generate the failed to open alarm.
   // 
   // If the timer reaches zero, and the valve is closing, generate the failed to close alarm
   // ▄▄▄▄▄▄▄▄▄▄▄▄▄▄▄▄▄▄▄▄▄▄▄▄▄▄▄▄▄▄▄▄▄▄▄▄▄▄▄▄▄▄▄▄
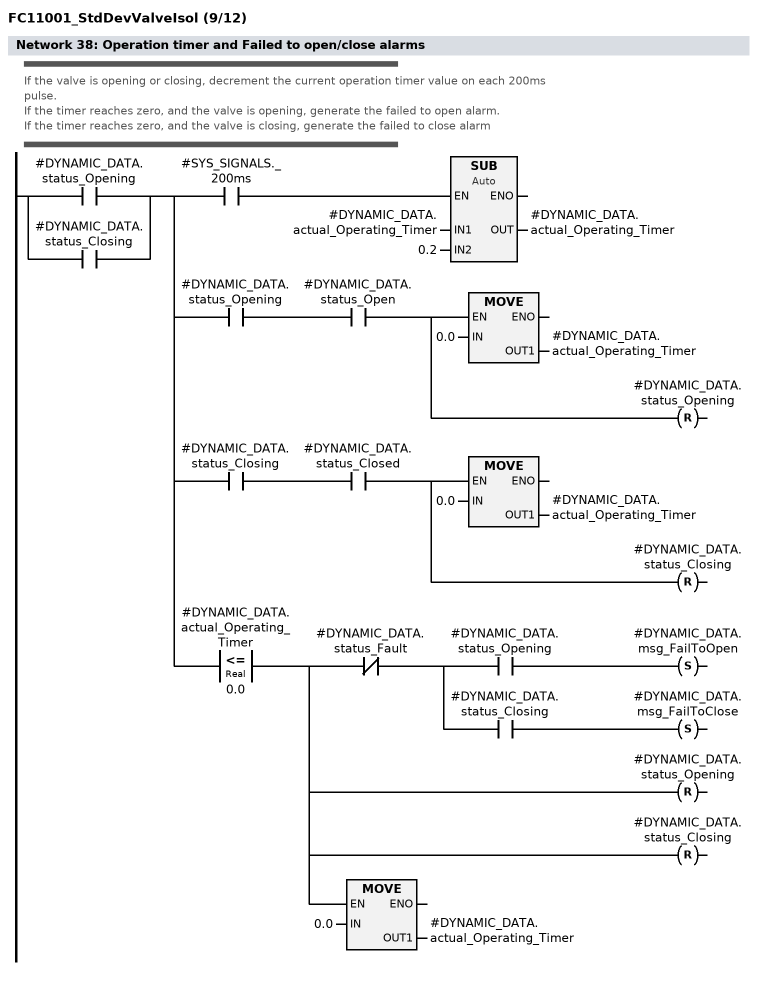
   RUNG wire#powerrail
      Contact( #DYNAMIC_DATA.status_Opening )
      wire#w1
      Contact( #SYS_SIGNALS._200ms )
      Sub(in1 := #DYNAMIC_DATA.actual_Operating_Timer, in2 := 0.2, out => #DYNAMIC_DATA.actual_Operating_Timer)
   END_RUNG
   RUNG wire#powerrail
      Contact( #DYNAMIC_DATA.status_Closing )
   END_RUNG wire#w1
   RUNG wire#w1
      Contact( #DYNAMIC_DATA.status_Opening )
      Contact( #DYNAMIC_DATA.status_Open )
      wire#w2
      Move(in := 0.0, out1 => #DYNAMIC_DATA.actual_Operating_Timer)
   END_RUNG
   RUNG wire#w2
      R_Coil( #DYNAMIC_DATA.status_Opening )
   END_RUNG
   RUNG wire#w1
      Contact( #DYNAMIC_DATA.status_Closing )
      Contact( #DYNAMIC_DATA.status_Closed )
      wire#w3
      Move(in := 0.0, out1 => #DYNAMIC_DATA.actual_Operating_Timer)
   END_RUNG
   RUNG wire#w3
      R_Coil( #DYNAMIC_DATA.status_Closing )
   END_RUNG
   RUNG wire#w1
      { S7_Templates := "SrcType := Real" } LE_Contact(in1 := #DYNAMIC_DATA.actual_Operating_Timer, in2 := 0.0)
      wire#w4
      I_Contact( #DYNAMIC_DATA.status_Fault )
      wire#w5
      Contact( #DYNAMIC_DATA.status_Opening )
      S_Coil( #DYNAMIC_DATA.msg_FailToOpen )
   END_RUNG
   RUNG wire#w5
      Contact( #DYNAMIC_DATA.status_Closing )
      S_Coil( #DYNAMIC_DATA.msg_FailToClose )
   END_RUNG
   RUNG wire#w4
      R_Coil( #DYNAMIC_DATA.status_Opening )
   END_RUNG
   RUNG wire#w4
      R_Coil( #DYNAMIC_DATA.status_Closing )
   END_RUNG
   RUNG wire#w4
      Move(in := 0.0, out1 => #DYNAMIC_DATA.actual_Operating_Timer)
   END_RUNG
   // the same network as SCL:
   #_w1 := #DYNAMIC_DATA.status_Opening OR #DYNAMIC_DATA.status_Closing;
   IF #_w1 AND #SYS_SIGNALS._200ms THEN
       #DYNAMIC_DATA.actual_Operating_Timer := #DYNAMIC_DATA.actual_Operating_Timer - 0.2;
   END_IF;
   IF #_w1 AND #DYNAMIC_DATA.status_Opening AND #DYNAMIC_DATA.status_Open THEN
       #DYNAMIC_DATA.actual_Operating_Timer := 0.0;
       #DYNAMIC_DATA.status_Opening := FALSE;
   END_IF;
   IF #_w1 AND #DYNAMIC_DATA.status_Closing AND #DYNAMIC_DATA.status_Closed THEN
       #DYNAMIC_DATA.actual_Operating_Timer := 0.0;
       #DYNAMIC_DATA.status_Closing := FALSE;
   END_IF;
   #_w2 := #_w1 AND (#DYNAMIC_DATA.actual_Operating_Timer <= 0.0);
   #_w3 := #_w2 AND NOT #DYNAMIC_DATA.status_Fault;
   IF #_w3 AND #DYNAMIC_DATA.status_Opening THEN #DYNAMIC_DATA.msg_FailToOpen := TRUE; END_IF;
   IF #_w3 AND #DYNAMIC_DATA.status_Closing THEN #DYNAMIC_DATA.msg_FailToClose := TRUE; END_IF;
   IF #_w2 THEN
       #DYNAMIC_DATA.status_Opening := FALSE;
       #DYNAMIC_DATA.status_Closing := FALSE;
       #DYNAMIC_DATA.actual_Operating_Timer := 0.0;
   END_IF;
END_REGION

REGION Network 39: Calculate last operation timer value
   // ▀▀▀▀▀▀▀▀▀▀▀▀▀▀▀▀▀▀▀▀▀▀▀▀▀▀▀▀▀▀▀▀▀▀▀▀▀▀▀▀▀▀▀▀
   // Stores that last good operation timer elapsed time, this is the elapsed value of the 
   // actual_Operating_Timer when the valve achieved the correct position. The result is subtracted
   // from the TIME_OPENING/CLOSING_MAX value to give the true time to achieve position. The result
   // is stored in actual_Last_Op_Time
   // 
   // If the valve were opening, then actual_Last_Op_Time is calculated as follows:
   // 
   // ┌─────────────────────────────────┐
   // │actual_Last_Op_Time = TIME_OPENING_MAX ─ actual_Operating_Timer   │
   // └─────────────────────────────────┘
   // 
   // If the valve were closing, then actual_Last_Op_Time is calculated as follows:
   // 
   // ┌─────────────────────────────────┐
   // │actual_Last_Op_Time = TIME_CLOSING_MAX ─ actual_Operating_Timer   │
   // └─────────────────────────────────┘
   // 
   // If the valve either fails to open or fails to close,  then actual_Last_Op_Time is set to -1.0 to 
   // indicate a fault state.
   // ▄▄▄▄▄▄▄▄▄▄▄▄▄▄▄▄▄▄▄▄▄▄▄▄▄▄▄▄▄▄▄▄▄▄▄▄▄▄▄▄▄▄▄▄
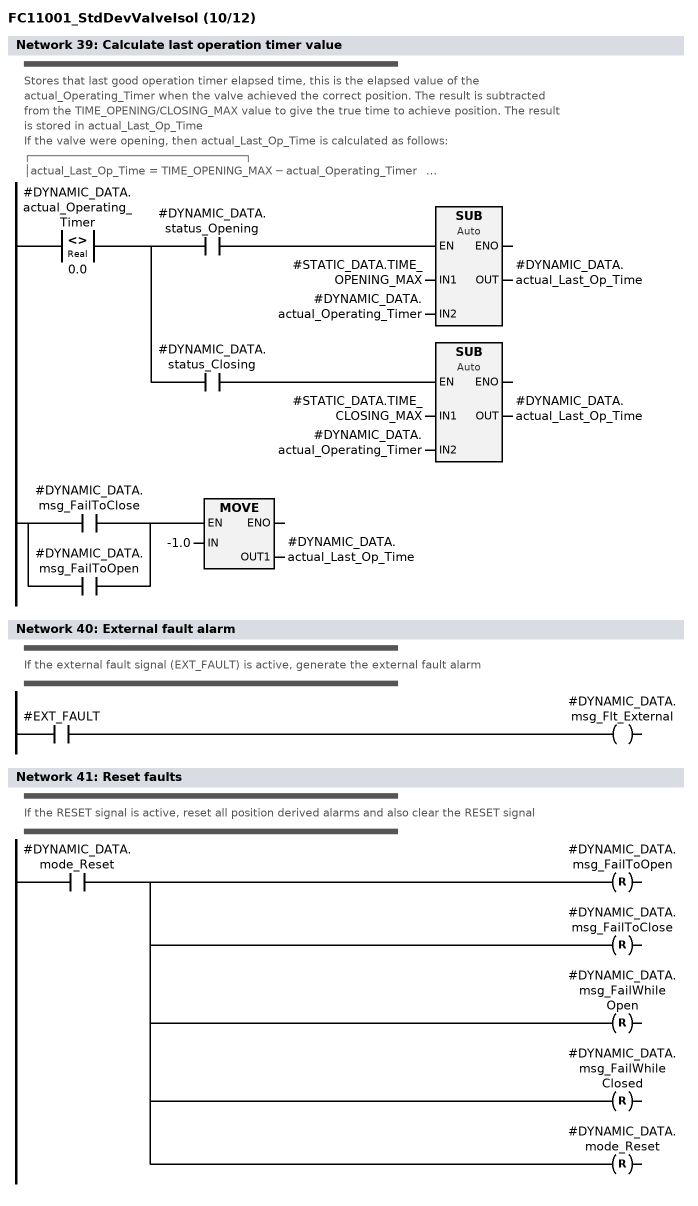
   RUNG wire#powerrail
      { S7_Templates := "SrcType := Real" } NE_Contact(in1 := #DYNAMIC_DATA.actual_Operating_Timer, in2 := 0.0)
      wire#w1
      Contact( #DYNAMIC_DATA.status_Opening )
      Sub(in1 := #STATIC_DATA.TIME_OPENING_MAX, in2 := #DYNAMIC_DATA.actual_Operating_Timer, out => #DYNAMIC_DATA.actual_Last_Op_Time)
   END_RUNG
   RUNG wire#w1
      Contact( #DYNAMIC_DATA.status_Closing )
      Sub(in1 := #STATIC_DATA.TIME_CLOSING_MAX, in2 := #DYNAMIC_DATA.actual_Operating_Timer, out => #DYNAMIC_DATA.actual_Last_Op_Time)
   END_RUNG
   RUNG wire#powerrail
      Contact( #DYNAMIC_DATA.msg_FailToClose )
      wire#w2
      Move(in := -1.0, out1 => #DYNAMIC_DATA.actual_Last_Op_Time)
   END_RUNG
   RUNG wire#powerrail
      Contact( #DYNAMIC_DATA.msg_FailToOpen )
   END_RUNG wire#w2
   // the same network as SCL:
   #_w1 := #DYNAMIC_DATA.actual_Operating_Timer <> 0.0;
   IF #_w1 AND #DYNAMIC_DATA.status_Opening THEN
       #DYNAMIC_DATA.actual_Last_Op_Time := #STATIC_DATA.TIME_OPENING_MAX - #DYNAMIC_DATA.actual_Operating_Timer;
   END_IF;
   IF #_w1 AND #DYNAMIC_DATA.status_Closing THEN
       #DYNAMIC_DATA.actual_Last_Op_Time := #STATIC_DATA.TIME_CLOSING_MAX - #DYNAMIC_DATA.actual_Operating_Timer;
   END_IF;
   IF #DYNAMIC_DATA.msg_FailToClose OR #DYNAMIC_DATA.msg_FailToOpen THEN
       #DYNAMIC_DATA.actual_Last_Op_Time := -1.0;
   END_IF;
END_REGION

REGION Network 40: External fault alarm
   // ▀▀▀▀▀▀▀▀▀▀▀▀▀▀▀▀▀▀▀▀▀▀▀▀▀▀▀▀▀▀▀▀▀▀▀▀▀▀▀▀▀▀▀▀
   // If the external fault signal (EXT_FAULT) is active, generate the external fault alarm
   // ▄▄▄▄▄▄▄▄▄▄▄▄▄▄▄▄▄▄▄▄▄▄▄▄▄▄▄▄▄▄▄▄▄▄▄▄▄▄▄▄▄▄▄▄
   RUNG wire#powerrail
      Contact( #EXT_FAULT )
      Coil( #DYNAMIC_DATA.msg_Flt_External )
   END_RUNG
   // the same network as SCL:
   #DYNAMIC_DATA.msg_Flt_External := #EXT_FAULT;
END_REGION

REGION Network 41: Reset faults
   // ▀▀▀▀▀▀▀▀▀▀▀▀▀▀▀▀▀▀▀▀▀▀▀▀▀▀▀▀▀▀▀▀▀▀▀▀▀▀▀▀▀▀▀▀
   // If the RESET signal is active, reset all position derived alarms and also clear the RESET signal
   // ▄▄▄▄▄▄▄▄▄▄▄▄▄▄▄▄▄▄▄▄▄▄▄▄▄▄▄▄▄▄▄▄▄▄▄▄▄▄▄▄▄▄▄▄
   RUNG wire#powerrail
      Contact( #DYNAMIC_DATA.mode_Reset )
      wire#w1
      R_Coil( #DYNAMIC_DATA.msg_FailToOpen )
   END_RUNG
   RUNG wire#w1
      R_Coil( #DYNAMIC_DATA.msg_FailToClose )
   END_RUNG
   RUNG wire#w1
      R_Coil( #DYNAMIC_DATA.msg_FailWhileOpen )
   END_RUNG
   RUNG wire#w1
      R_Coil( #DYNAMIC_DATA.msg_FailWhileClosed )
   END_RUNG
   RUNG wire#w1
      R_Coil( #DYNAMIC_DATA.mode_Reset )
   END_RUNG
   // the same network as SCL:
   IF #DYNAMIC_DATA.mode_Reset THEN
       #DYNAMIC_DATA.msg_FailToOpen := FALSE;
       #DYNAMIC_DATA.msg_FailToClose := FALSE;
       #DYNAMIC_DATA.msg_FailWhileOpen := FALSE;
       #DYNAMIC_DATA.msg_FailWhileClosed := FALSE;
       #DYNAMIC_DATA.mode_Reset := FALSE;
   END_IF;
END_REGION

